(* POU STP, ST *)
PROGRAM STP
VAR
	LSL100A_MixerFloatSensor AT %I* : BOOL;
	LSH100A_MixerFloatSensor AT %I* : BOOL;
	LSH101A_EQFloatSensor AT %I* : BOOL;
	LSHH101A_EQFloatSensor AT %I* : BOOL;
	LSL101A_EQFloatSensor AT %I* : BOOL;
	LSH105A1_StreamLineFlow AT %I* : BOOL;
	LSHH105A2_StreamLineOverflow AT %I* : BOOL;
	LSL103A_SBRFloatSensor AT %I* : BOOL;
	LSHH103A_SBRFloatSensor AT %I* : BOOL;
	LSH103A_SBRFloatSensor AT %I* : BOOL;
	F100_FanStatus AT %I* : BOOL;
	D100_DoorPanelStatus AT %I* : BOOL;
	LSD101A_EQFloatSensorDry AT %I* : BOOL;
	LSD103A_SBRFloatSensorDry AT %I* : BOOL;
	XV101A1_SolenoidValveSpray_OpenStat AT %I* : BOOL;
	XV101A2_SolenoidValveSpray_OpenStat AT %I* : BOOL;
	XV102A1_ContinuosValveWater_OpenStat AT %I* : BOOL;
	XV100A1_GritRemovalValve_OpenStat AT %I* : BOOL;
	XV100A2_GritRemovalValve_OpenStat AT %I* : BOOL;
	PS101A1_Penstock_OpenStat AT %I* : BOOL;
	PS101A2_Penstock_OpenStat AT %I* : BOOL;
	PS101A1_Penstock_CloseStat AT %I* : BOOL;
	PS101A2_Penstock_CloseStat AT %I* : BOOL;
	XV101A1_SolenoidValveSpray_CloseStat AT %I* : BOOL;
	XV101A2_SolenoidValveSpray_CloseStat AT %I* : BOOL;
	XV102A1_ContinuosValveWater_CloseStat AT %I* : BOOL;
	XV100A1_GritRemovalValve_CloseStat AT %I* : BOOL;
	XV100A2_GritRemovalValve_CloseStat AT %I* : BOOL;
	M101A1_EQMixer_OverloadStat AT %I* : BOOL;
	M101A1_EQMixer_IncompleteStat AT %I* : BOOL;
	M101A2_EQMixer_OverloadStat AT %I* : BOOL;
	M101A2_EQMixer_IncompleteStat AT %I* : BOOL;
	P101A1_EQPump_OverloadStat AT %I* : BOOL;
	P101A1_EQPump_IncompleteStat AT %I* : BOOL;
	P101A2_EQPump_OverloadStat AT %I* : BOOL;
	P101A2_EQPump_IncompleteStat AT %I* : BOOL;
	PS101A1_Penstock_TripStat AT %I* : BOOL;
	PS101A2_Penstock_TripStat AT %I* : BOOL;
	F101A1_FineScr_OverloadStat AT %I* : BOOL;
	F101A2_FineScr_OverloadStat AT %I* : BOOL;
	C102A_ScreeningConveyer_OverloadStat AT %I* : BOOL;
	C101A_ScreeningCompactor_OverloadStat AT %I* : BOOL;
	C103A_GritClassifier_OverloadStat AT %I* : BOOL;
	P102A1_SBRTransferPump_OverloadStat AT %I* : BOOL;
	P102A1_SBRTransferPump_IncompleteStat AT %I* : BOOL;
	P102A2_SBRTransferPump_OverloadStat AT %I* : BOOL;
	P102A2_SBRTransferPump_IncompleteStat AT %I* : BOOL;
	M101A1_EQMixer_LocalRemoteStat AT %I* : BOOL;
	M101A2_EQMixer_LocalRemoteStat AT %I* : BOOL;
	P101A1_EQPump_LocalRemoteStat AT %I* : BOOL;
	P101A2_EQPump_LocalRemoteStat AT %I* : BOOL;
	F101A1_FineScr_LocalRemoteStat AT %I* : BOOL;
	F101A2_FineScr_LocalRemoteStat AT %I* : BOOL;
	C102A_ScreenConveyer_LocalRemoteStat AT %I* : BOOL;
	C101A_ScreenCompactor_LocalRemoteStat AT %I* : BOOL;
	C103A_GritClasifier_LocalRemoteStat AT %I* : BOOL;
	P102A1_SBRTransferPump_LocalRemoteStat AT %I* : BOOL;
	P102A2_SBRTransferPump_LocalRemoteStat AT %I* : BOOL;
	PS101A1_Penstock_LocalRemoteStat AT %I* : BOOL;
	PS101A2_Penstock_LocalRemoteStat AT %I* : BOOL;
	M101A1_EQMixer_RunStat AT %I* : BOOL;
	M101A2_EQMixer_RunStat AT %I* : BOOL;
	P101A1_EQPump_RunStat AT %I* : BOOL;
	P101A2_EQPump_RunStat AT %I* : BOOL;
	F101A1_FineScr_RunStat AT %I* : BOOL;
	F101A2_FineScr_RunStat AT %I* : BOOL;
	C102A_ScreenConveyer_RunStat AT %I* : BOOL;
	C101A_ScreenCompactor_RunStat AT %I* : BOOL;
	C103A_GritClasifier_RunStat AT %I* : BOOL;
	P102A1_SBRTransferPump_RunStat AT %I* : BOOL;
	P102A2_SBRTransferPump_RunStat AT %I* : BOOL;
	M101A1_EQMixer_EStopStat AT %I* : BOOL;
	M101A2_EQMixer_EStopStat AT %I* : BOOL;
	P101A1_EQPump_EStopStat AT %I* : BOOL;
	P101A2_EQPump_EStopStat AT %I* : BOOL;
	F101A1_FineScr_EStopStat AT %I* : BOOL;
	F101A2_FineScr_EStopStat AT %I* : BOOL;
	C102A_ScreenConveyer_EStopStat AT %I* : BOOL;
	C101A_ScreenCompactor_EStopStat AT %I* : BOOL;
	C103A_GritClasifier_EStopStat AT %I* : BOOL;
	P102A1_SBRTransferPump_EStopStat AT %I* : BOOL;
	P102A2_SBRTransferPump_EStopStat AT %I* : BOOL;
	B101A1_AirBlower_OverloadStat AT %I* : BOOL;
	B101A1_AirBlower_IncompleteStat AT %I* : BOOL;
	B101A2_AirBlower_OverloadStat AT %I* : BOOL;
	B101A2_AirBlower_IncompleteStat AT %I* : BOOL;
	B101A1_AirBlower_LocalRemoteStat AT %I* : BOOL;
	B101A2_AirBlower_LocalRemoteStat AT %I* : BOOL;
	B101A1_AirBlower_OnOffStat AT %I* : BOOL;
	B101A2_AirBlower_OnOffStat AT %I* : BOOL;
	B101A1_AirBlower_EStopStat AT %I* : BOOL;
	B101A2_AirBlower_EStopStat AT %I* : BOOL;
	XV101A1_SolenoidValveSpray_OpenCmd AT %Q* : BOOL;
	XV101A2_SolenoidValveSpray_OpenCmd AT %Q* : BOOL;
	XV102A1_ContinuosValveWater_OpenCmd AT %Q* : BOOL;
	F101A1_FineScr_RunCmd AT %Q* : BOOL;
	F101A2_FineScr_RunCmd AT %Q* : BOOL;
	C102A_ScreenConveyer_RunCmd AT %Q* : BOOL;
	C101A_ScreenCompactor_RunCmd AT %Q* : BOOL;
	C103A_GritClasifier_RunCmd AT %Q* : BOOL;
	PS101A1_Penstock_OpenCmd AT %Q* : BOOL;
	PS101A1_Penstock_CloseCmd AT %Q* : BOOL;
	PS101A2_Penstock_OpenCmd AT %Q* : BOOL;
	PS101A2_Penstock_CloseCmd AT %Q* : BOOL;
	XV100A1_GritRemovalValve_OpenCmd AT %Q* : BOOL;
	XV100A2_GritRemovalValve_OpenCmd AT %Q* : BOOL;
	P101A1_EQPump_RunCmd AT %Q* : BOOL;
	P101A2_EQPump_RunCmd AT %Q* : BOOL;
	M101A1_EQMixer_RunCmd AT %Q* : BOOL;
	M101A2_EQMixer_RunCmd AT %Q* : BOOL;
	B101A1_AirBlower_RunCmd AT %Q* : BOOL;
	B101A2_AirBlower_RunCmd AT %Q* : BOOL;
	P102A1_SBRTransferPump_RunCmd AT %Q* : BOOL;
	P102A2_SBRTransferPump_RunCmd AT %Q* : BOOL;
	AUX101A_EQFloatSensor_AlarmS1 AT %Q* : BOOL;
	AUX104A_SBRFloatSensor_AlarmS1 AT %Q* : BOOL;
	AUX105A_StreamSensorOverflow_AlarmS1 AT %Q* : BOOL;
	AUX106_CommonAlarm AT %Q* : BOOL;
	AUX107_PLCRunStat AT %Q* : BOOL;
	LSL100B_MixerFloatSensor AT %I* : BOOL;
	LSH100B_MixerFloatSensor AT %I* : BOOL;
	LSH101B_EQFloatSensor AT %I* : BOOL;
	LSHH101B_EQFloatSensor AT %I* : BOOL;
	LSL101B_EQFloatSensor AT %I* : BOOL;
	LSH105B1_StreamLineFlow AT %I* : BOOL;
	LSHH105B2_StreamLineOverflow AT %I* : BOOL;
	LSH103B_SBRFloatSensor AT %I* : BOOL;
	LSHH103B_SBRFloatSensor AT %I* : BOOL;
	LSL103B_SBRFloatSensor AT %I* : BOOL;
	LSD101B_EQFloatSensorDry AT %I* : BOOL;
	LSD103B_SBRFloatSensorDry AT %I* : BOOL;
	XV101B1_SolenoidValveSpray_OpenStat AT %I* : BOOL;
	XV101B2_SolenoidValveSpray_OpenStat AT %I* : BOOL;
	XV102B1_ContinuosValveWater_OpenStat AT %I* : BOOL;
	XV100B1_GritRemovalValve_OpenStat AT %I* : BOOL;
	XV100B2_GritRemovalValve_OpenStat AT %I* : BOOL;
	PS101B1_Penstock_OpenStat AT %I* : BOOL;
	PS101B2_Penstock_OpenStat AT %I* : BOOL;
	PS101B1_Penstock_CloseStat AT %I* : BOOL;
	PS101B2_Penstock_CloseStat AT %I* : BOOL;
	XV101B1_SolenoidValveSpray_CloseStat AT %I* : BOOL;
	XV101B2_SolenoidValveSpray_CloseStat AT %I* : BOOL;
	XV102B1_ContinuosValveWater_CloseStat AT %I* : BOOL;
	XV100B1_GritRemovalValve_CloseStat AT %I* : BOOL;
	XV100B2_GritRemovalValve_CloseStat AT %I* : BOOL;
	M101B1_EQMixer_OverloadStat AT %I* : BOOL;
	M101B1_EQMixer_IncompleteStat AT %I* : BOOL;
	M101B2_EQMixer_OverloadStat AT %I* : BOOL;
	M101B2_EQMixer_IncompleteStat AT %I* : BOOL;
	P101B1_EQPump_OverloadStat AT %I* : BOOL;
	P101B1_EQPump_IncompleteStat AT %I* : BOOL;
	P101B2_EQPump_OverloadStat AT %I* : BOOL;
	P101B2_EQPump_IncompleteStat AT %I* : BOOL;
	PS101B1_Penstock_TripStat AT %I* : BOOL;
	PSB101B2_Penstock_TripStat AT %I* : BOOL;
	F101B1_FineScr_OverloadStat AT %I* : BOOL;
	F101B2_FineScr_OverloadStat AT %I* : BOOL;
	C102B_ScreeningConveyer_OverloadStat AT %I* : BOOL;
	C101B_ScreeningCompactor_OverloadStat AT %I* : BOOL;
	C103B_GritClassifier_OverloadStat AT %I* : BOOL;
	P102B1_SBRTransferPump_OverloadStat AT %I* : BOOL;
	P102B1_SBRTransferPump_IncompleteStat AT %I* : BOOL;
	P102B2_SBRTransferPump_OverloadStat AT %I* : BOOL;
	P102B2_SBRTransferPump_IncompleteStat AT %I* : BOOL;
	M101B1_EQMixer_LocalRemoteStat AT %I* : BOOL;
	M101B2_EQMixer_LocalRemoteStat AT %I* : BOOL;
	P101B1_EQPump_LocalRemoteStat AT %I* : BOOL;
	P101B2_EQPump_LocalRemoteStat AT %I* : BOOL;
	F101B1_FineScr_LocalRemoteStat AT %I* : BOOL;
	F101B2_FineScr_LocalRemoteStat AT %I* : BOOL;
	C102B_ScreenConveyer_LocalRemoteStat AT %I* : BOOL;
	C101B_ScreenCompactor_LocalRemoteStat AT %I* : BOOL;
	C103B_GritClasifiier_LocalRemoteStat AT %I* : BOOL;
	P102B1_SBRTransferPump_LocalRemoteStat AT %I* : BOOL;
	P102B2_SBRTransferPump_LocalRemoteStat AT %I* : BOOL;
	PS101B1_Penstock_LocalRemoteStat AT %I* : BOOL;
	PS101B2_Penstock_LocalRemoteStat AT %I* : BOOL;
	M101B1_EQMixer_RunStat AT %I* : BOOL;
	M101B2_EQMixer_RunStat AT %I* : BOOL;
	P101B1_EQPump_RunStat AT %I* : BOOL;
	P101B2_EQPump_RunStat AT %I* : BOOL;
	F101B1_FineScr_RunStat AT %I* : BOOL;
	F101B2_FineScr_RunStat AT %I* : BOOL;
	C102B_ScreenConveyer_RunStat AT %I* : BOOL;
	C101B_ScreenCompactor_RunStat AT %I* : BOOL;
	C103B_GritClasifier_RunStat AT %I* : BOOL;
	P102B1_SBRTransferPump_RunStat AT %I* : BOOL;
	P102B2_SBRTransferPump_RunStat AT %I* : BOOL;
	M101B1_EQMixer_EStopStat AT %I* : BOOL;
	M101B2_EQMixer_EStopStat AT %I* : BOOL;
	P101B1_EQPump_EStopStat AT %I* : BOOL;
	P101B2_EQPump_EStopStat AT %I* : BOOL;
	F101B1_FineScr_EStopStat AT %I* : BOOL;
	F101B2_FineScr_EStopStat AT %I* : BOOL;
	C102B_ScreenConveyer_EStopStat AT %I* : BOOL;
	C101B_ScreenCompactor_EStopStat AT %I* : BOOL;
	C103B_GritClasifier_EStopStat AT %I* : BOOL;
	P102B1_SBRTransferPump_EStopStat AT %I* : BOOL;
	P102B2_SBRTransferPump_EStopStat AT %I* : BOOL;
	VE801A_SuctionFan_OnOffStat AT %I* : BOOL;
	P802A_CirculationPump_OnOffStat AT %I* : BOOL;
	P803A_CirculationPump_OnOffStat AT %I* : BOOL;
	P804A_CirculationPump_OnOffStat AT %I* : BOOL;
	P805A1_H2S04Pump_OnOffStat AT %I* : BOOL;
	P805A2_H2S04Pump_OnOffStat AT %I* : BOOL;
	P806A1_NAOHPump_OnOffStat AT %I* : BOOL;
	P806A2_NAOHPump_OnOffStat AT %I* : BOOL;
	P807A1_NAOCLPump_OnOffStat AT %I* : BOOL;
	P807A2_NAOCLPump_OnOffStat AT %I* : BOOL;
	VE801A_SuctionFan_OverloadStat AT %I* : BOOL;
	P802A_CirculationPump_OverloadStat AT %I* : BOOL;
	P803A_CirculationPump_OverloadStat AT %I* : BOOL;
	P804A_CirculationPump_OverloadStat AT %I* : BOOL;
	P805A1_H2S04Pump_OverloadStat AT %I* : BOOL;
	P805A2_H2S04Pump_OverloadStat AT %I* : BOOL;
	P806A1_NAOHPump_OverloadStat AT %I* : BOOL;
	P806A2_NAOHPump_OverloadStat AT %I* : BOOL;
	P807A1_NAOCLPump_OverloadStat AT %I* : BOOL;
	P807A2_NAOCLPump_OverloadStat AT %I* : BOOL;
	VE801A_SuctionFan_EStopStat AT %I* : BOOL;
	P802A_CirculationPump_EStopStat AT %I* : BOOL;
	P803A_CirculationPump_EStopStat AT %I* : BOOL;
	P804A_CirculationPump_EStopStat AT %I* : BOOL;
	P805A1_H2S04Pump_EStopStat AT %I* : BOOL;
	P805A2_H2S04Pump_EStopStat AT %I* : BOOL;
	P806A1_NAOHPump_EStopStat AT %I* : BOOL;
	P806A2_NAOHPump_EStopStat AT %I* : BOOL;
	P807A1_NAOCLPump_EStopStat AT %I* : BOOL;
	P807A2_NAOCLPump_EStopStat AT %I* : BOOL;
	XV101B1_SolenoidValveSpray_OpenCmd AT %Q* : BOOL;
	XV101B2_SolenoidValveSpray_OpenCmd AT %Q* : BOOL;
	XV102B1_ContinuosValveWater_OpenCmd AT %Q* : BOOL;
	F101B1_FineScr_RunCmd AT %Q* : BOOL;
	F101B2_FineScr_RunCmd AT %Q* : BOOL;
	C102B_ScreenConveyer_RunCmd AT %Q* : BOOL;
	C101B_ScreenCompactor_RunCmd AT %Q* : BOOL;
	C103B_GritClasifier_RunCmd AT %Q* : BOOL;
	PS101B1_Penstock_OpenCmd AT %Q* : BOOL;
	PS101B1_Penstock_CloseCmd AT %Q* : BOOL;
	PS101B2_Penstock_OpenCmd AT %Q* : BOOL;
	PS101B2_Penstock_CloseCmd AT %Q* : BOOL;
	XV100B1_GritRemovalValve_OpenCmd AT %Q* : BOOL;
	XV100B2_GritRemovalValve_OpenCmd AT %Q* : BOOL;
	P101B1_EQPump_RunCmd AT %Q* : BOOL;
	P101B2_EQPump_RunCmd AT %Q* : BOOL;
	M101B1_EQMixer_RunCmd AT %Q* : BOOL;
	M101B2_EQMixer_RunCmd AT %Q* : BOOL;
	P102B1_SBRTransferPump_RunCmd AT %Q* : BOOL;
	P102B2_SBRTransferPump_RunCmd AT %Q* : BOOL;
	AUX101B_EQFloatSensor_AlarmS2 AT %Q* : BOOL;
	AUX104B_SBRFloatSensor_AlarmS2 AT %Q* : BOOL;
	AUX105B_StreamSensorOverflow_AlarmS2 AT %Q* : BOOL;
	F200A_FanStatus AT %I* : BOOL;
	D200A_DoorPanelStatus AT %I* : BOOL;
	XV261A_DecanterR1_OverloadStat AT %I* : BOOL;
	XV262A_DecanterR2_OverloadStat AT %I* : BOOL;
	XV263A_DecanterR3_OverloadStat AT %I* : BOOL;
	XV264A_DecanterR4_OverloadStat AT %I* : BOOL;
	M200A1A_MixerR1_RunStat AT %I* : BOOL;
	M200A1B_MixerR1_RunStat AT %I* : BOOL;
	M200A1C_MixerR1_RunStat AT %I* : BOOL;
	M200A2A_MixerR2_RunStat AT %I* : BOOL;
	M200A2B_MixerR2_RunStat AT %I* : BOOL;
	M200A2C_MixerR2_RunStat AT %I* : BOOL;
	M200A3A_MixerR3_RunStat AT %I* : BOOL;
	M200A3B_MixerR3_RunStat AT %I* : BOOL;
	M200A3C_MixerR3_RunStat AT %I* : BOOL;
	M200A4A_MixerR4_RunStat AT %I* : BOOL;
	M200A4B_MixerR4_RunStat AT %I* : BOOL;
	M200A4C_MixerR4_RunStat AT %I* : BOOL;
	B201A1_AirBlowerS1_RunStat AT %I* : BOOL;
	B201A2_AirBlowerS1_RunStat AT %I* : BOOL;
	B201A3_AirBlowerS1_RunStat AT %I* : BOOL;
	M200A1A_MixerR1_LocalRemoteStat AT %I* : BOOL;
	M200A1B_MixerR1_LocalRemoteStat AT %I* : BOOL;
	M200A1C_MixerR1_LocalRemoteStat AT %I* : BOOL;
	M200A2A_MixerR2_LocalRemoteStat AT %I* : BOOL;
	M200A2B_MixerR2_LocalRemoteStat AT %I* : BOOL;
	M200A2C_MixerR2_LocalRemoteStat AT %I* : BOOL;
	M200A3A_MixerR3_LocalRemoteStat AT %I* : BOOL;
	M200A3B_MixerR3_LocalRemoteStat AT %I* : BOOL;
	M200A3C_MixerR3_LocalRemoteStat AT %I* : BOOL;
	M200A4A_MixerR4_LocalRemoteStat AT %I* : BOOL;
	M200A4B_MixerR4_LocalRemoteStat AT %I* : BOOL;
	M200A4C_MixerR4_LocalRemoteStat AT %I* : BOOL;
	B201A1_AirBlowerS1_LocalRemoteStat AT %I* : BOOL;
	B201A2_AirBlowerS1_LocalRemoteStat AT %I* : BOOL;
	B201A3_AirBlowerS1_LocalRemoteStat AT %I* : BOOL;
	XV261A_DecanterR1_LocalRemoteStat AT %I* : BOOL;
	XV262A_DecanterR2_LocalRemoteStat AT %I* : BOOL;
	XV263A_DecanterR3_LocalRemoteStat AT %I* : BOOL;
	XV264A_DecanterR4_LocalRemoteStat AT %I* : BOOL;
	P201A1_DesludgePumpS1_LocalRemoteStat AT %I* : BOOL;
	P201A2_DesludgePumpS1_LocalRemoteStat AT %I* : BOOL;
	P201A1_DesludgePumpS1_RunStat AT %I* : BOOL;
	P201A2_DesludgePumpS1_RunStat AT %I* : BOOL;
	M200A1A_MixerR1_OverloadStat AT %I* : BOOL;
	M200A1A_MixerR1_IncompleteStat AT %I* : BOOL;
	M200A1B_MixerR1_OverloadStat AT %I* : BOOL;
	M200A1B_MixerR1_IncompleteStat AT %I* : BOOL;
	M200A1C_MixerR1_OverloadStat AT %I* : BOOL;
	M200A1C_MixerR1_IncompleteStat AT %I* : BOOL;
	M200A2A_MixerR2_OverloadStat AT %I* : BOOL;
	M200A2A_MixerR2_IncompleteStat AT %I* : BOOL;
	M200A2B_MixerR2_OverloadStat AT %I* : BOOL;
	M200A2B_MixerR2_IncompleteStat AT %I* : BOOL;
	M200A2C_MixerR2_OverloadStat AT %I* : BOOL;
	M200A2C_MixerR2_IncompleteStat AT %I* : BOOL;
	M200A3A_MixerR3_OverloadStat AT %I* : BOOL;
	M200A3A_MixerR3_IncompleteStat AT %I* : BOOL;
	M200A3B_MixerR3_OverloadStat AT %I* : BOOL;
	M200A3B_MixerR3_IncompleteStat AT %I* : BOOL;
	M200A3C_MixerR3_OverloadStat AT %I* : BOOL;
	M200A3C_MixerR3_IncompleteStat AT %I* : BOOL;
	M200A4A_MixerR4_OverloadStat AT %I* : BOOL;
	M200A4A_MixerR4_IncompleteStat AT %I* : BOOL;
	M200A4B_MixerR4_OverloadStat AT %I* : BOOL;
	M200A4B_MixerR4_IncompleteStat AT %I* : BOOL;
	M200A4C_MixerR4_OverloadStat AT %I* : BOOL;
	M200A4C_MixerR4_IncompleteStat AT %I* : BOOL;
	B201A1_AirBlowerS1_OverloadStat AT %I* : BOOL;
	B201A1_AirBlowerS1_IncompleteStat AT %I* : BOOL;
	B201A2_AirBlowerS1_OverloadStat AT %I* : BOOL;
	B201A2_AirBlowerS1_IncompleteStat AT %I* : BOOL;
	B201A3_AirBlowerS1_OverloadStat AT %I* : BOOL;
	B201A3_AirBlowerS1_IncompleteStat AT %I* : BOOL;
	P201A1_DesludgePumpS1_OverloadStatus AT %I* : BOOL;
	P201A2_DesludgePumpS1_OverloadStatus AT %I* : BOOL;
	M200A1A_MixerR1_EStopStat AT %I* : BOOL;
	M200A1B_MixerR1_EStopStat AT %I* : BOOL;
	M200A1C_MixerR1_EStopStat AT %I* : BOOL;
	M200A2A_MixerR2_EStopStat AT %I* : BOOL;
	M200A2B_MixerR2_EStopStat AT %I* : BOOL;
	M200A2C_MixerR2_EStopStat AT %I* : BOOL;
	M200A3A_MixerR3_EStopStat AT %I* : BOOL;
	M200A3B_MixerR3_EStopStat AT %I* : BOOL;
	M200A3C_MixerR3_EStopStat AT %I* : BOOL;
	M200A4A_MixerR3_EStopStat AT %I* : BOOL;
	M200A4B_MixerR3_EStopStat AT %I* : BOOL;
	M200A4C_MixerR3_EStopStat AT %I* : BOOL;
	B201A1_AirBlowerS1_EStopStat AT %I* : BOOL;
	B201A2_AirBlowerS1_EStopStat AT %I* : BOOL;
	B201A3_AirBlowerS1_EStopStat AT %I* : BOOL;
	XV261A_DecanterR1_EStopStat AT %I* : BOOL;
	XV262A_DecanterR2_EStopStat AT %I* : BOOL;
	XV263A_DecanterR3_EStopStat AT %I* : BOOL;
	XV264A_DecanterR4_EStopStat AT %I* : BOOL;
	P201A1_DesludgePumpS1_EStopStat AT %I* : BOOL;
	P201A2_DesludgePumpS1_EStopStat AT %I* : BOOL;
	XV261A_DecanterR1_FwdStat AT %I* : BOOL;
	XV262A_DecanterR2_FwdStat AT %I* : BOOL;
	XV263A_DecanterR3_FwdStat AT %I* : BOOL;
	XV264A_DecanterR4_FwdStat AT %I* : BOOL;
	XV261A_DecanterR1_RvsStat AT %I* : BOOL;
	XV262A_DecanterR2_RvsStat AT %I* : BOOL;
	XV263A_DecanterR3_RvsStat AT %I* : BOOL;
	XV264A_DecanterR4_RvsStat AT %I* : BOOL;
	FT100A_FlowTotalizerS1 : REAL;
	FT100A_FlowTotalizerS1_ScaledValue AT %I*:INT;
	M200A1A_MixerR1_RunCmd AT %Q* : BOOL;
	M200A1B_MixerR1_RunCmd AT %Q* : BOOL;
	M200A1C_MixerR1_RunCmd AT %Q* : BOOL;
	M200A2A_MixerR2_RunCmd AT %Q* : BOOL;
	M200A2B_MixerR2_RunCmd AT %Q* : BOOL;
	M200A2C_MixerR2_RunCmd AT %Q* : BOOL;
	M200A3A_MixerR3_RunCmd AT %Q* : BOOL;
	M200A3B_MixerR3_RunCmd AT %Q* : BOOL;
	M200A3C_MixerR3_RunCmd AT %Q* : BOOL;
	M200A4A_MixerR4_RunCmd AT %Q* : BOOL;
	M200A4B_MixerR4_RunCmd AT %Q* : BOOL;
	M200A4C_MixerR4_RunCmd AT %Q* : BOOL;
	XV261A_DecanterR1_FwdCmd AT %Q* : BOOL;
	XV262A_DecanterR2_FwdCmd AT %Q* : BOOL;
	XV263A_DecanterR3_FwdCmd AT %Q* : BOOL;
	XV264A_DecanterR4_FwdCmd AT %Q* : BOOL;
	XV261A_DecanterR1_RvsCmd AT %Q* : BOOL;
	XV262A_DecanterR2_RvsCmd AT %Q* : BOOL;
	XV263A_DecanterR3_RvsCmd AT %Q* : BOOL;
	XV264A_DecanterR4_RvsCmd AT %Q* : BOOL;
	B201A1_AirBlowerS1_RunCmd AT %Q* : BOOL;
	B201A2_AirBlowerS1_RunCmd AT %Q* : BOOL;
	B201A3_AirBlowerS1_RunCmd AT %Q* : BOOL;
	P201A1_DesludgePump_RunCmd AT %Q* : BOOL;
	P201A2_DesludgePump_RunCmd AT %Q* : BOOL;
	AUXA1_ReactorS1R1_OpsStat AT %Q* : BOOL;
	AUXA2_ReactorS1R2_OpsStat AT %Q* : BOOL;
	AUXA3_ReactorS1R3_OpsStat AT %Q* : BOOL;
	AUXA4_ReactorS1R4_OpsStat AT %Q* : BOOL;
	AUXB1_ReactorS2R1_OpsStat AT %Q* : BOOL;
	AUXB2_ReactorS2R2_OpsStat AT %Q* : BOOL;
	AUXB3_ReactorS2R3_OpsStat AT %Q* : BOOL;
	AUXB4_ReactorS2R4_OpsStat AT %Q* : BOOL;
	AUXA5_BlowerS1R1 AT %Q* : BOOL;
	AUXA6_BlowerS1R2 AT %Q* : BOOL;
	AUXA7_BlowerS1R3 AT %Q* : BOOL;
	AUXB5_BlowerS2R1 AT %Q* : BOOL;
	AUXB6_BlowerS2R2 AT %Q* : BOOL;
	AUXB7_BlowerS2R3 AT %Q* : BOOL;
	AUX201_CommonAlarm AT %Q* : BOOL;
	AUX202_PLCRunStat AT %Q* : BOOL;
	F200B_FanStatus AT %I* : BOOL;
	D200B_DoorPanelStatus AT %I* : BOOL;
	XV261B_DecanterR1_OverloadStat AT %I* : BOOL;
	XV262B_DecanterR2_OverloadStat AT %I* : BOOL;
	XV263B_DecanterR3_OverloadStat AT %I* : BOOL;
	XV264B_DecanterR4_OverloadStat AT %I* : BOOL;
	M200B1A_MixerR1_RunStat AT %I* : BOOL;
	M200B1B_MixerR1_RunStat AT %I* : BOOL;
	M200B1C_MixerR1_RunStat AT %I* : BOOL;
	M200B2A_MixerR2_RunStat AT %I* : BOOL;
	M200B2B_MixerR2_RunStat AT %I* : BOOL;
	M200B2C_MixerR2_RunStat AT %I* : BOOL;
	M200B3A_MixerR3_RunStat AT %I* : BOOL;
	M200B3B_MixerR3_RunStat AT %I* : BOOL;
	M200B3C_MixerR3_RunStat AT %I* : BOOL;
	M200B4A_MixerR4_RunStat AT %I* : BOOL;
	M200B4B_MixerR4_RunStat AT %I* : BOOL;
	M200B4C_MixerR4_RunStat AT %I* : BOOL;
	B201B1_AirBlowerS2_RunStat AT %I* : BOOL;
	B201B2_AirBlowerS2_RunStat AT %I* : BOOL;
	B201B3_AirBlowerS2_RunStat AT %I* : BOOL;
	M200B1A_MixerR1_LocalRemoteStat AT %I* : BOOL;
	M200B1B_MixerR1_LocalRemoteStat AT %I* : BOOL;
	M200B1C_MixerR1_LocalRemoteStat AT %I* : BOOL;
	M200B2A_MixerR2_LocalRemoteStat AT %I* : BOOL;
	M200B2B_MixerR2_LocalRemoteStat AT %I* : BOOL;
	M200B2C_MixerR2_LocalRemoteStat AT %I* : BOOL;
	M200B3A_MixerR3_LocalRemoteStat AT %I* : BOOL;
	M200B3B_MixerR3_LocalRemoteStat AT %I* : BOOL;
	M200B3C_MixerR3_LocalRemoteStat AT %I* : BOOL;
	M200B4A_MixerR4_LocalRemoteStat AT %I* : BOOL;
	M200B4B_MixerR4_LocalRemoteStat AT %I* : BOOL;
	M200B4C_MixerR4_LocalRemoteStat AT %I* : BOOL;
	B201B1_AirBlowerS2_LocalRemoteStat AT %I* : BOOL;
	B201B2_AirBlowerS2_LocalRemoteStat AT %I* : BOOL;
	B201B3_AirBlowerS2_LocalRemoteStat AT %I* : BOOL;
	XV261B_DecanterR1_LocalRemoteStat AT %I* : BOOL;
	XV262B_DecanterR2_LocalRemoteStat AT %I* : BOOL;
	XV263B_DecanterR3_LocalRemoteStat AT %I* : BOOL;
	XV264B_DecanterR4_LocalRemoteStat AT %I* : BOOL;
	P201B1_DesludgePumpS2_LocalRemoteStat AT %I* : BOOL;
	P201B2_DesludgePumpS2_LocalRemoteStat AT %I* : BOOL;
	P201B1_DesludgePumpS2_RunStat AT %I* : BOOL;
	P201B2_DesludgePumpS2_RunStat AT %I* : BOOL;
	M200B1A_MixerR1_OverloadStat AT %I* : BOOL;
	M200B1A_MixerR1_IncompleteStat AT %I* : BOOL;
	M200B1B_MixerR1_OverloadStat AT %I* : BOOL;
	M200B1B_MixerR1_IncompleteStat AT %I* : BOOL;
	M200B1C_MixerR1_OverloadStat AT %I* : BOOL;
	M200B1C_MixerR1_IncompleteStat AT %I* : BOOL;
	M200B2A_MixerR2_OverloadStat AT %I* : BOOL;
	M200B2A_MixerR2_IncompleteStat AT %I* : BOOL;
	M200B2B_MixerR2_OverloadStat AT %I* : BOOL;
	M200B2B_MixerR2_IncompleteStat AT %I* : BOOL;
	M200B2C_MixerR2_OverloadStat AT %I* : BOOL;
	M200B2C_MixerR2_IncompleteStat AT %I* : BOOL;
	M200B3A_MixerR3_OverloadStat AT %I* : BOOL;
	M200B3A_MixerR2_IncompleteStat AT %I* : BOOL;
	M200B3B_MixerR3_OverloadStat AT %I* : BOOL;
	M200B3B_MixerR3_IncompleteStat AT %I* : BOOL;
	M200B3C_MixerR3_OverloadStat AT %I* : BOOL;
	M200B3C_MixerR3_IncompleteStat AT %I* : BOOL;
	M200B4A_MixerR4_OverloadStat AT %I* : BOOL;
	M200B4A_MixerR4_IncompleteStat AT %I* : BOOL;
	M200B4B_MixerR4_OverloadStat AT %I* : BOOL;
	M200B4B_MixerR4_IncompleteStat AT %I* : BOOL;
	M200B4C_MixerR4_OverloadStat AT %I* : BOOL;
	M200B4C_MixerR4_IncompleteStat AT %I* : BOOL;
	B201B1_AirBlowerS2_OverloadStat AT %I* : BOOL;
	B201B1_AirBlowerS2_IncompleteStat AT %I* : BOOL;
	B201B2_AirBlowerS2_OverloadStat AT %I* : BOOL;
	B201B2_AirBlowerS2_IncompleteStat AT %I* : BOOL;
	B201B3_AirBlowerS2_OverloadStat AT %I* : BOOL;
	B201B3_AirBlowerS2_IncompleteStat AT %I* : BOOL;
	P201B1_DesludgePumpS2_OverloadStat AT %I* : BOOL;
	P201B2_DesludgePumpS2_OverloadStat AT %I* : BOOL;
	M200B1A_MixerR1_EStopStat AT %I* : BOOL;
	M200B1B_MixerR1_EStopStat AT %I* : BOOL;
	M200B1C_MixerR1_EStopStat AT %I* : BOOL;
	M200B2A_MixerR2_EStopStat AT %I* : BOOL;
	M200B2B_MixerR2_EStopStat AT %I* : BOOL;
	M200B2C_MixerR2_EStopStat AT %I* : BOOL;
	M200B3A_MixerR3_EStopStat AT %I* : BOOL;
	M200B3B_MixerR3_EStopStat AT %I* : BOOL;
	M200B3C_MixerR3_EStopStat AT %I* : BOOL;
	M200B4A_MixerR4_EStopStat AT %I* : BOOL;
	M200B4B_MixerR4_EStopStat AT %I* : BOOL;
	M200B4C_MixerR4_EStopStat AT %I* : BOOL;
	B201B1_AirBlowerS2_EStopStat AT %I* : BOOL;
	B201B2_AirBlowerS2_EStopStat AT %I* : BOOL;
	B201B3_AirBlowerS2_EStopStat AT %I* : BOOL;
	XV261B_DecanterR1_EStopStat AT %I* : BOOL;
	XV262B_DecanterR2_EStopStat AT %I* : BOOL;
	XV263B_DecanterR3_EStopStat AT %I* : BOOL;
	XV264B_DecanterR4_EStopStat AT %I* : BOOL;
	P201B1_DesludgePumpS2_EStopStat AT %I* : BOOL;
	P201B2_DesludgePumpS2_EStopStat AT %I* : BOOL;
	XV261B_DecanterR1_FwdStat AT %I* : BOOL;
	XV262B_DecanterR2_FwdStat AT %I* : BOOL;
	XV263B_DecanterR3_FwdStat AT %I* : BOOL;
	XV264B_DecanterR4_FwdStat AT %I* : BOOL;
	XV261B_DecanterR1_RvsStat AT %I* : BOOL;
	XV262B_DecanterR2_RvsStat AT %I* : BOOL;
	XV263B_DecanterR3_RvsStat AT %I* : BOOL;
	XV264B_DecanterR4_RvsStat AT %I* : BOOL;
	FT100B_FlowTotalizerS2 : REAL;
	FT100B_FlowTotalizerS2_ScaledValue AT %I*:INT;
	M200B1A_MixerR1_RunCmd AT %Q* : BOOL;
	M200B1B_MixerR1_RunCmd AT %Q* : BOOL;
	M200B1C_MixerR1_RunCmd AT %Q* : BOOL;
	M200B2A_MixerR2_RunCmd AT %Q* : BOOL;
	M200B2B_MixerR2_RunCmd AT %Q* : BOOL;
	M200B2C_MixerR2_RunCmd AT %Q* : BOOL;
	M200B3A_MixerR3_RunCmd AT %Q* : BOOL;
	M200B3B_MixerR3_RunCmd AT %Q* : BOOL;
	M200B3C_MixerR3_RunCmd AT %Q* : BOOL;
	M200B4A_MixerR4_RunCmd AT %Q* : BOOL;
	M200B4B_MixerR4_RunCmd AT %Q* : BOOL;
	M200B4C_MixerR4_RunCmd AT %Q* : BOOL;
	XV261B_DecanterR1_FwdCmd AT %Q* : BOOL;
	XV262B_DecanterR2_FwdCmd AT %Q* : BOOL;
	XV263B_DecanterR3_FwdCmd AT %Q* : BOOL;
	XV264B_DecanterR4_FwdCmd AT %Q* : BOOL;
	XV261B_DecanterR1_RvsCmd AT %Q* : BOOL;
	XV262B_DecanterR2_RvsCmd AT %Q* : BOOL;
	XV263B_DecanterR3_RvsCmd AT %Q* : BOOL;
	XV264B_DecanterR4_RvsCmd AT %Q* : BOOL;
	B201B1_AirBlowerS2_RunCmd AT %Q* : BOOL;
	B201B2_AirBlowerS2_RunCmd AT %Q* : BOOL;
	B201B3_AirBlowerS2_RunCmd AT %Q* : BOOL;
	P201B1_DesludgePumpS2_RunCmd AT %Q* : BOOL;
	P201B2_DesludgePumpS2_RunCmd AT %Q* : BOOL;
	LSH201A1_LevelSensorR1 AT %I* : BOOL;
	LSH201A2_LevelSensorR2 AT %I* : BOOL;
	LSH201A3_LevelSensorR3 AT %I* : BOOL;
	LSH201A4_LevelSensorR4 AT %I* : BOOL;
	OPR1A_ReactorStatus AT %I* : BOOL;
	OPR2A_ReactorStatus AT %I* : BOOL;
	OPR3A_ReactorStatus AT %I* : BOOL;
	OPR4A_ReactorStatus AT %I* : BOOL;
	D201A_DoorPanelStatus AT %I* : BOOL;
	F201A_FanStatus AT %I* : BOOL;
	HR201A1_DecantHighLevelR1 AT %I* : BOOL;
	LR201A1_DecantLowLevelR1 AT %I* : BOOL;
	HR201A2_DecantHighLevelR2 AT %I* : BOOL;
	LR201A2_DecantLowLevelR2 AT %I* : BOOL;
	HR201A3_DecantHighLevelR3 AT %I* : BOOL;
	LR201A3_DecantLowLevelR3 AT %I* : BOOL;
	HR201A4_DecantHighLevelR4 AT %I* : BOOL;
	LR201A4_DecantLowLevelR4 AT %I* : BOOL;
	XV205A_SBRValveR1_OpenStat AT %I* : BOOL;
	XV206A_SBRValveR2_OpenStat AT %I* : BOOL;
	XV207A_SBRValveR3_OpenStat AT %I* : BOOL;
	XV208A_SBRValveR4_OpenStat AT %I* : BOOL;
	XV201A_AirBlowerValveR1_OpenStat AT %I* : BOOL;
	XV202A_AirBlowerValveR2_OpenStat AT %I* : BOOL;
	XV203A_AirBlowerValveR3_OpenStat AT %I* : BOOL;
	XV204A_AirBlowerValveR4_OpenStat AT %I* : BOOL;
	XV221A_LimeValveR1_OpenStat AT %I* : BOOL;
	XV222A_LimeValveR2_OpenStat AT %I* : BOOL;
	XV223A_LimeValveR3_OpenStat AT %I* : BOOL;
	XV224A_LimeValveR4_OpenStat AT %I* : BOOL;
	XV211A_AlumValveR1_OpenStat AT %I* : BOOL;
	XV212A_AlumValveR2_OpenStat AT %I* : BOOL;
	XV213A_AlumValveR3_OpenStat AT %I* : BOOL;
	XV214A_AlumValveR4_OpenStat AT %I* : BOOL;
	XV205A_SBRValveR1_CloseStat AT %I* : BOOL;
	XV206A_SBRValveR2_CloseStat AT %I* : BOOL;
	XV207A_SBRValveR3_CloseStat AT %I* : BOOL;
	XV208A_SBRValveR4_CloseStat AT %I* : BOOL;
	XV201A_AirBlowerValveR1_CloseStat AT %I* : BOOL;
	XV202A_AirBlowerValveR2_CloseStat AT %I* : BOOL;
	XV203A_AirBlowerValveR3_CloseStat AT %I* : BOOL;
	XV204A_AirBlowerValveR4_CloseStat AT %I* : BOOL;
	XV221A_LimeValveR1_CloseStat AT %I* : BOOL;
	XV222A_LimeValveR2_CloseStat AT %I* : BOOL;
	XV223A_LimeValveR3_CloseStat AT %I* : BOOL;
	XV224A_LimeValveR4_CloseStat AT %I* : BOOL;
	XV211A_AlumValveR1_CloseStat AT %I* : BOOL;
	XV212A_AlumValveR2_CloseStat AT %I* : BOOL;
	XV213A_AlumValveR3_CloseStat AT %I* : BOOL;
	XV214A_AlumValveR4_CloseStat AT %I* : BOOL;
	XV241A_SludgeValveR1_CloseStat AT %I* : BOOL;
	XV242A_SludgeValveR2_CloseStat AT %I* : BOOL;
	XV243A_SludgeValveR3_CloseStat AT %I* : BOOL;
	XV244A_SludgeValveR4_CloseStat AT %I* : BOOL;
	XV241A_SludgeValveR1_OpenStat AT %I* : BOOL;
	XV242A_SludgeValveR2_OpenStat AT %I* : BOOL;
	XV243A_SludgeValveR3_OpenStat AT %I* : BOOL;
	XV244A_SludgeValveR4_OpenStat AT %I* : BOOL;
	D0201A4_DOProfilesR4 : REAL;
	D0201A4_DOProfilesR4_ScaledValue AT %I*:INT;
	DO201A1_DOProfilesR1:REAL;
	DO201A1_DOProfilesR1_ScaledValue AT %I*:INT;
	DO201A2_DOProfilesR2 :REAL;
	DO201A2_DOProfilesR2_ScaledValue AT %I*:INT;
	DO201A3_DOProfilesR3 :REAL;
	DO201A3_DOProfilesR3_ScaledValue AT %I*:INT;
	PHT201A1_pHlevelR1 : REAL;
	PHT201A1_pHlevelR1_ScaledValue AT %I*:INT;
	PHT201A2_pHlevelR2 : REAL;
	PHT201A2_pHlevelR2_ScaledValue AT %I*:INT;
	PHT201A3_pHlevelR3 : REAL;
	PHT201A3_pHlevelR3_ScaledValue AT %I*:INT;
	PHT201A4_pHlevelR4 : REAL;
	PHT201A4_pHlevelR4_ScaledValue AT %I*:INT;
	XV205A_SBRValveR1_OpenCmd AT %Q* : BOOL;
	XV206A_SBRValveR2_OpenCmd AT %Q* : BOOL;
	XV207A_SBRValveR3_OpenCmd AT %Q* : BOOL;
	XV208A_SBRValveR4_OpenCmd AT %Q* : BOOL;
	XV201A_AirBlowerValveR1_OpenCmd AT %Q* : BOOL;
	XV202A_AirBlowerValveR2_OpenCmd AT %Q* : BOOL;
	XV203A_AirBlowerValveR3_OpenCmd AT %Q* : BOOL;
	XV204A_AirBlowerValveR4_OpenCmd AT %Q* : BOOL;
	XV221A_LimeValveR1_OpenCmd AT %Q* : BOOL;
	XV222A_LimeValveR2_OpenCmd AT %Q* : BOOL;
	XV223A_LimeValveR3_OpenCmd AT %Q* : BOOL;
	XV224A_LimeValveR4_OpenCmd AT %Q* : BOOL;
	XV211A_AlumValveR1_OpenCmd AT %Q* : BOOL;
	XV212A_AlumValveR2_OpenCmd AT %Q* : BOOL;
	XV213A_AlumValveR3_OpenCmd AT %Q* : BOOL;
	XV214A_AlumValveR4_OpenCmd AT %Q* : BOOL;
	XV241A_SludgeValveR1_OpenCmd AT %Q* : BOOL;
	XV242A_SludgeValveR2_OpenCmd AT %Q* : BOOL;
	XV243A_SludgeValveR3_OpenCmd AT %Q* : BOOL;
	XV244A_SludgeValveR4_OpenCmd AT %Q* : BOOL;
	XV241A_SludgeValveR1_CloseCmd AT %Q* : BOOL;
	XV242A_SludgeValveR2_CloseCmd AT %Q* : BOOL;
	XV243A_SludgeValveR3_CloseCmd AT %Q* : BOOL;
	XV244A_SludgeValveR4_CloseCmd AT %Q* : BOOL;
	XV205A_SBRValveR1_CloseCmd AT %Q* : BOOL;
	XV206A_SBRValveR2_CloseCmd AT %Q* : BOOL;
	XV207A_SBRValveR3_CloseCmd AT %Q* : BOOL;
	XV208A_SBRValveR4_CloseCmd AT %Q* : BOOL;
	XV201A_AirBlowerValveR1_CloseCmd AT %Q* : BOOL;
	XV202A_AirBlowerValveR2_CloseCmd AT %Q* : BOOL;
	XV203A_AirBlowerValveR3_CloseCmd AT %Q* : BOOL;
	XV204A_AirBlowerValveR4_CloseCmd AT %Q* : BOOL;
	XV221A_LimeValveR1_CloseCmd AT %Q* : BOOL;
	XV222A_LimeValveR2_CloseCmd AT %Q* : BOOL;
	XV223A_LimeValveR3_CloseCmd AT %Q* : BOOL;
	XV224A_LimeValveR4_CloseCmd AT %Q* : BOOL;
	XV211A_AlumValveR1_CloseCmd AT %Q* : BOOL;
	XV212A_AlumValveR2_CloseCmd AT %Q* : BOOL;
	XV213A_AlumValveR3_CloseCmd AT %Q* : BOOL;
	XV214A_AlumValveR4_CloseCmd AT %Q* : BOOL;
	OPR1AON_ReactorR1_OnlineCmd AT %Q* : BOOL;
	OPR2AON_ReactorR2_OnlineCmd AT %Q* : BOOL;
	OPR3AON_ReactorR3_OnlineCmd AT %Q* : BOOL;
	OPR4AON_ReactorR4_OnlineCmd AT %Q* : BOOL;
	OPR1AOFF_ReactorR1_OfflineCmd AT %Q* : BOOL;
	OPR2AOFF_ReactorR2_OfflineCmd AT %Q* : BOOL;
	OPR3AOFF_ReactorR3_OfflineCmd AT %Q* : BOOL;
	OPR4AOFF_ReactorR4_OfflineCmd AT %Q* : BOOL;
	OPR1ASW_ReactorR1_SwitchCmd AT %Q* : BOOL;
	OPR2ASW_ReactorR2_SwitchCmd AT %Q* : BOOL;
	OPR3ASW_ReactorR3_SwitchCmd AT %Q* : BOOL;
	OPR4ASW_ReactorR4_SwitchCmd AT %Q* : BOOL;
	AUX402_PLCRunStat AT %Q* : BOOL;
	AUX401_CommonAlarm AT %Q* : BOOL;
	LSH201B1_LevelSensorR1 AT %I* : BOOL;
	LSH201B2_LevelSensorR2 AT %I* : BOOL;
	LSH201B3_LevelSensorR3 AT %I* : BOOL;
	LSH201B4_LevelSensorR4 AT %I* : BOOL;
	OPR1B_ReactorStatus AT %I* : BOOL;
	OPR2B_ReactorStatus AT %I* : BOOL;
	OPR3B_ReactorStatus AT %I* : BOOL;
	OPR4B_ReactorStatus AT %I* : BOOL;
	D201B_DoorPanelStatus AT %I* : BOOL;
	F201B_FanStatus AT %I* : BOOL;
	HR201B1_DecantHighLevelR1 AT %I* : BOOL;
	LR201B1_DecantLowLevelR1 AT %I* : BOOL;
	HR201B2_DecantHighLevelR2 AT %I* : BOOL;
	LR201B2_DecantLowLevelR2 AT %I* : BOOL;
	HR201B3_DecantHighLevelR3 AT %I* : BOOL;
	HR201B4_DecantHighLevelR4 AT %I* : BOOL;
	LR201B3_DecantLowLevelR3 AT %I* : BOOL;
	LR201B4_DecantLowLevelR4 AT %I* : BOOL;
	XV205B_SBRValveR1_OpenStat AT %I* : BOOL;
	XV206B_SBRValveR2_OpenStat AT %I* : BOOL;
	XV207B_SBRValveR3_OpenStat AT %I* : BOOL;
	XV208B_SBRValveR4_OpenStat AT %I* : BOOL;
	XV201B_AirBlowerValveR1_OpenStat AT %I* : BOOL;
	XV202B_AirBlowerValveR2_OpenStat AT %I* : BOOL;
	XV203B_AirBlowerValveR3_OpenStat AT %I* : BOOL;
	XV204B_AirBlowerValveR4_OpenStat AT %I* : BOOL;
	XV221B_LimeValveR1_OpenStat AT %I* : BOOL;
	XV222B_LimeValveR2_OpenStat AT %I* : BOOL;
	XV223B_LimeValveR3_OpenStat AT %I* : BOOL;
	XV224B_LimeValveR4_OpenStat AT %I* : BOOL;
	XV211B_AlumValveR1_OpenStat AT %I* : BOOL;
	XV212B_AlumValveR2_OpenStat AT %I* : BOOL;
	XV213B_AlumValveR3_OpenStat AT %I* : BOOL;
	XV214B_AlumValveR4_OpenStat AT %I* : BOOL;
	XV205B_SBRValveR1_CloseStat AT %I* : BOOL;
	XV206B_SBRValveR2_CloseStat AT %I* : BOOL;
	XV207B_SBRValveR3_CloseStat AT %I* : BOOL;
	XV208B_SBRValveR4_CloseStat AT %I* : BOOL;
	XV201B_AirBlowerValveR1_CloseStat AT %I* : BOOL;
	XV202B_AirBlowerValveR2_CloseStat AT %I* : BOOL;
	XV203B_AirBlowerValveR3_CloseStat AT %I* : BOOL;
	XV204B_AirBlowerValveR4_CloseStat AT %I* : BOOL;
	XV221B_LimeValveR1_CloseStat AT %I* : BOOL;
	XV222B_LimeValveR2_CloseStat AT %I* : BOOL;
	XV223B_LimeValveR3_CloseStat AT %I* : BOOL;
	XV224B_LimeValveR4_CloseStat AT %I* : BOOL;
	XV211B_AlumValveR1_CloseStat AT %I* : BOOL;
	XV212B_AlumValveR2_CloseStat AT %I* : BOOL;
	XV213B_AlumValveR3_CloseStat AT %I* : BOOL;
	XV214B_AlumValveR4_CloseStat AT %I* : BOOL;
	XV241B_SludgeValveR1_CloseStat AT %I* : BOOL;
	XV242B_SludgeValveR2_CloseStat AT %I* : BOOL;
	XV243B_SludgeValveR3_CloseStat AT %I* : BOOL;
	XV244B_SludgeValveR4_CloseStat AT %I* : BOOL;
	XV241B_SludgeValveR1_OpenStat AT %I* : BOOL;
	XV242B_SludgeValveR2_OpenStat AT %I* : BOOL;
	XV243B_SludgeValveR3_OpenStat AT %I* : BOOL;
	XV244B_SludgeValveR4_OpenStat AT %I* : BOOL;
	DO201B1_DOProfilesR1: REAL;
	DO201B1_DOProfilesR1_ScaledValue AT%I*:INT;
	DO201B2_DOProfilesR2: REAL;
	DO201B2_DOProfilesR2_ScaledValue AT %I*:INT;
	DO201B3_DOProfilesR3 : REAL;
	DO201B3_DOProfilesR3_ScaledValue AT %I*:INT;
	D0201B4_DOProfilesR4 : REAL;
	D0201B4_DOProfilesR4_ScaledValue AT %I*:INT;
	PHT201B1_pHlevelR1 : REAL;
	PHT201B1_pHlevelR1_ScaledValue AT%I*:INT;
	PHT201B2_pHlevelR2 : REAL;
	PHT201B2_pHlevelR2_ScaledValue AT %I*  :INT;
	PHT201B3_pHlevelR3  : REAL;
	PHT201B3_pHlevelR3_ScaledValue AT %I*:INT;
	PHT201B4_pHlevelR4  : REAL;
	PHT201B4_pHlevelR4_ScaledValue AT %I*:INT;
	XV205B_SBRValveR1_OpenCmd AT %Q* : BOOL;
	XV206B_SBRValveR2_OpenCmd AT %Q* : BOOL;
	XV207B_SBRValveR3_OpenCmd AT %Q* : BOOL;
	XV208B_SBRValveR4_OpenCmd AT %Q* : BOOL;
	XV202B_AirBlowerValveR2_OpenCmd AT %Q* : BOOL;
	XV201B_AirBlowerValveR1_OpenCmd AT %Q* : BOOL;
	XV204B_AirBlowerValveR4_OpenCmd AT %Q* : BOOL;
	XV203B_AirBlowerValveR3_OpenCmd AT %Q* : BOOL;
	XV221B_LimeValveR1_OpenCmd AT %Q* : BOOL;
	XV222B_LimeValveR2_OpenCmd AT %Q* : BOOL;
	XV223B_LimeValveR3_OpenCmd AT %Q* : BOOL;
	XV224B_LimeValveR4_OpenCmd AT %Q* : BOOL;
	XV211B_AlumValveR1_OpenCmd AT %Q* : BOOL;
	XV212B_AlumValveR2_OpenCmd AT %Q* : BOOL;
	XV213B_AlumValveR3_OpenCmd AT %Q* : BOOL;
	XV214B_AlumValveR4_OpenCmd AT %Q* : BOOL;
	XV241B_SludgeValveR1_OpenCmd AT %Q* : BOOL;
	XV242B_SludgeValveR2_OpenCmd AT %Q* : BOOL;
	XV243B_SludgeValveR3_OpenCmd AT %Q* : BOOL;
	XV244B_SludgeValveR4_OpenCmd AT %Q* : BOOL;
	XV241B_SludgeValveR1_CloseCmd AT %Q* : BOOL;
	XV242B_SludgeValveR2_CloseCmd AT %Q* : BOOL;
	XV243B_SludgeValveClosedR3_CloseCmd AT %Q* : BOOL;
	XV244B_SludgeValveR4_CloseCmd AT %Q* : BOOL;
	XV205B_SBRValveR1_CloseCmd AT %Q* : BOOL;
	XV206B_SBRValveR2_CloseCmd AT %Q* : BOOL;
	XV207B_SBRValveR3_CloseCmd AT %Q* : BOOL;
	XV208B_SBRValveR4_CloseCmd AT %Q* : BOOL;
	XV201B_AirBlowerValveR1_CloseCmd AT %Q* : BOOL;
	XV202B_AirBlowerValveR2_CloseCmd AT %Q* : BOOL;
	XV203B_AirBlowerValveR3_CloseCmd AT %Q* : BOOL;
	XV204B_AirBlowerValveR4_CloseCmd AT %Q* : BOOL;
	XV221B_LimeValveR1_CloseCmd AT %Q* : BOOL;
	XV222B_LimeValveR2_CloseCmd AT %Q* : BOOL;
	XV223B_LimeValveR3_CloseCmd AT %Q* : BOOL;
	XV224B_LimeValveR4_CloseCmd AT %Q* : BOOL;
	XV211B_AlumValveR1_CloseCmd AT %Q* : BOOL;
	XV212B_AlumValveR2_CloseCmd AT %Q* : BOOL;
	XV213B_AlumValveR3_CloseCmd AT %Q* : BOOL;
	XV214B_AlumValveR4_CloseCmd AT %Q* : BOOL;
	OPR1BON_ReactorR1_OnlineCmd AT %Q* : BOOL;
	OPR2BON_ReactorR2_OnlineCmd AT %Q* : BOOL;
	OPR3BON_ReactorR3_OnlineCmd AT %Q* : BOOL;
	OPR4BON_ReactorR4_OnlineCmd AT %Q* : BOOL;
	OPR1BOFF_ReactorR1_OfflineCmd AT %Q* : BOOL;
	OPR2BOFF_ReactorR2_OfflineCmd AT %Q* : BOOL;
	OPR3BOFF_ReactorR3_OfflineCmd AT %Q* : BOOL;
	OPR4BOFF_ReactorR4_OfflineCmd AT %Q* : BOOL;
	OPR1BSW_ReactorR1_SwitchCmd AT %Q* : BOOL;
	OPR2BSW_ReactorR2_SwitchCmd AT %Q* : BOOL;
	OPR3BSW_ReactorR3_SwitchCmd AT %Q* : BOOL;
	OPR4BSW_ReactorR4_SwitchCmd AT %Q* : BOOL;
	AUX502_PLCRunStat AT %Q* : BOOL;
	AUX501_CommonAlarm AT %Q* : BOOL;
	LSHH210A_LimeTank1 AT %I* : BOOL;
	LSH210A_LimeTank1 AT %I* : BOOL;
	LSL210A_LimeTank1 AT %I* : BOOL;
	LSD210A_LimeTank1 AT %I* : BOOL;
	LSHH210B_LimeTank2 AT %I* : BOOL;
	LSH210B_LimeTank2 AT %I* : BOOL;
	LSL210B_LimeTank2 AT %I* : BOOL;
	LSD210B_LimeTank2 AT %I* : BOOL;
	LSHH210C_LimeTank3 AT %I* : BOOL;
	LSH210C_LimeTank3 AT %I* : BOOL;
	LSL210C_LimeTank3 AT %I* : BOOL;
	LSD210C_LimeTank3 AT %I* : BOOL;
	LSL351A_AlumTank1 AT %I* : BOOL;
	LSL351B_AlumTank2 AT %I* : BOOL;
	LSL351C_AlumTank3 AT %I* : BOOL;
	LSL351D_AlumTank4 AT %I* : BOOL;
	LSL355A_SodiumHypochloriteTank AT %I* : BOOL;
	LSL355B_SodiumHypochloriteTank AT %I* : BOOL;
	LSL355C_SodiumHypochloriteTank AT %I* : BOOL;
	LSL353A_CausticSodaTank AT %I* : BOOL;
	LSL353B_CausticSodaTank AT %I* : BOOL;
	LSHH301_EffluentSump AT %I* : BOOL;
	LSH301_EffluentSump AT %I* : BOOL;
	LSL301_EffluentSump AT %I* : BOOL;
	LSHH302_CollectionSump AT %I* : BOOL;
	LSH302_CollectionSump AT %I* : BOOL;
	LSL302_CollectionSump AT %I* : BOOL;
	LSH309A_ReUseWaterStorageTank1HIGH AT %I* : BOOL;
	LSH309B_ReUseWaterStorageTank2HIGH AT %I* : BOOL;
	XV251A_LimeSelectorTank_OpenStat AT %I* : BOOL;
	XV251B_LimeSelectorTank_OpenStat AT %I* : BOOL;
	XV251C_LimeSelectorTank_OpenStat AT %I* : BOOL;
	XV251A_LimeSelectorTank_CloseStat AT %I* : BOOL;
	XV251B_LimSelectorTank_CloseStat AT %I* : BOOL;
	XV251C_LimeSelectorTank_CloseStat AT %I* : BOOL;
	OPAlumA_AlumSelectorTank AT %I* : BOOL;
	OPAlumB_AlumSelectorTank AT %I* : BOOL;
	OPAlumC_AlumSelectorTank AT %I* : BOOL;
	OPAlumD_AlumSelectorTank AT %I* : BOOL;
	OPCausticA_CausticSodaSelectorTank1 AT %I* : BOOL;
	OPCausticB_CausticSodaSelectorTank2 AT %I* : BOOL;
	OPSodiumA_SodiumHypochloriteSelectorTank1 AT %I* : BOOL;
	OPSodiumB_SodiumHypochloriteSelectorTank2 AT %I* : BOOL;
	OPSodiumC_SodiumHypochloriteSelectorTank3 AT %I* : BOOL;
	P210A1_LimePumpS1_RunStat AT %I* : BOOL;
	P210A2_LimePumpS1S2_RunStat AT %I* : BOOL;
	P210A3_LimePumpS2_RunStat AT %I* : BOOL;
	P203A_LimeCirculationPump_RunStat AT %I* : BOOL;
	P203B_LimeCirculationPump_RunStat AT %I* : BOOL;
	P211A1_AlumPumpSBRS1_RunStat AT %I* : BOOL;
	P211A2_AlumPumpSBRS1_RunStat AT %I* : BOOL;
	P211B1_AlumPump1SBRS2_RunStat AT %I* : BOOL;
	P211B2_AlumPumpSBRS2_RunStat AT %I* : BOOL;
	P352A_AlumPumpTertiaryDosing_RunStat AT %I* : BOOL;
	P352B_AlumPumpTertiaryDosing_RunStat AT %I* : BOOL;
	XV210A1_LimeValveS1_OpenStat AT %I* : BOOL;
	XV201A2_LimeValveS2_OpenStat AT %I* : BOOL;
	XV210A1_LimeValveS1_CloseStat AT %I* : BOOL;
	XV201A2_LimeValveS2_CloseStat AT %I* : BOOL;
	P354A_CausticSodaPump_RunStat AT %I* : BOOL;
	P354B_CausticSodaPump_RunStat AT %I* : BOOL;
	P356A_SodiumHypochloritePumpChlorinetank_RunStat AT %I* : BOOL;
	P356B_SodiumHypochloritePumpChlorinetank_RunStat AT %I* : BOOL;
	P204A_SodiumHypochloritePumpDisinfectionTank_RunStat AT %I* : BOOL;
	P204B_SodiumHypochloritePumpDisinfectionTank_RunStat AT %I* : BOOL;
	M210A_LimeStirrer_OverloadStat AT %I* : BOOL;
	M210B_LimeStirrer_OverloadStat AT %I* : BOOL;
	M210C_LimeStirrer_OverloadStat AT %I* : BOOL;
	F300_FanStatus AT %I* : BOOL;
	D300_DoorPanelStatus AT %I* : BOOL;
	XV250A_LimeWaterIntakeTank_OpenStat AT %I* : BOOL;
	XV250B_LimeWaterIntakeTank_OpenStat AT %I* : BOOL;
	XV250C_LimeWaterIntakeTank_OpenStat AT %I* : BOOL;
	XV250A_LimeWaterIntakeTank_CloseStat AT %I* : BOOL;
	XV250B_LimeWaterIntakeTank_CloseStat AT %I* : BOOL;
	XV250C_LimeWaterIntakeTank_CloseStat AT %I* : BOOL;
	XV303A_LamellaSludgeDischarge_OpenStat AT %I* : BOOL;
	XV303B_LamellaSludgeDischarge_OpenStat AT %I* : BOOL;
	XV303C_LamellaSludgeDischarge_OpenStat AT %I* : BOOL;
	XV303D_LamellaSludgeDischarge_OpenStat AT %I* : BOOL;
	XV305_TertiaryTreatmentMainValve_OpenStat AT %I* : BOOL;
	XV303A_LamellaSludgeDischarge_CloseStat AT %I* : BOOL;
	XV303B_LamellaSludgeDischarge_CloseStat AT %I* : BOOL;
	XV303C_LamellaSludgeDischarge_CloseStat AT %I* : BOOL;
	XV303D_LamellaSludgeDischarge_CloseStat AT %I* : BOOL;
	XV305_TertiaryTreatmentMainValve_CloseStat AT %I* : BOOL;
	M210A_LimeStirrer_RunStat AT %I* : BOOL;
	M210B_LimeStirrer_RunStat AT %I* : BOOL;
	M210C_LimeStirrer_RunStat AT %I* : BOOL;
	M303A_Floculator_RunStat AT %I* : BOOL;
	M303B_Floculator_RunStat AT %I* : BOOL;
	M303C_Floculator_RunStat AT %I* : BOOL;
	M303D_Floculator_RunStat AT %I* : BOOL;
	P301A_EffluentTransferPump_RunStat AT %I* : BOOL;
	P301B_EffluentTransferPump_RunStat AT %I* : BOOL;
	AUX11_CascadeAerator_OnlineStat:BOOL;
	AUX12_ChlorineAnalyzer_OnlineStat:BOOL;
	P302A_CollectionPump_RunStat AT %I* : BOOL;
	P302B_CollectionPump_RunStat AT %I* : BOOL;
	K301A_AirCompressor_RunStat AT %I* : BOOL;
	K301B_AirCompressor_RunStat AT %I* : BOOL;
	P210A1_LimePumpS1_LocalRemoteStat AT %I* : BOOL;
	P210A2_LimePumpS1_LocalRemoteStat AT %I* : BOOL;
	P210A3_LimePumpS1_LocalRemoteStat AT %I* : BOOL;
	P203A_LimeCirculationPump1_LocalRemoteStat AT %I* : BOOL;
	P203B_LimeCirculationPump2_LocalRemoteStat AT %I* : BOOL;
	P211A1_AlumPumpSBRS1_LocalRemoteStat AT %I* : BOOL;
	P211A2_AlumPumpSBRS1_LocalRemoteStat AT %I* : BOOL;
	P211B1_AlumPumpSBRS2_LocalRemoteStat AT %I* : BOOL;
	P211B2_AlumPump2SBRS2_LocalRemoteStat AT %I* : BOOL;
	P352A_AlumPumpTertiaryDosing_LocalRemoteStat AT %I* : BOOL;
	P352B_AlumPumpTertiaryDosing_LocalRemoteStat AT %I* : BOOL;
	P354A_CausticSodaPump_LocalRemoteStat AT %I* : BOOL;
	P354B_CausticSodaPump_LocalRemoteStat AT %I* : BOOL;
	P356A_SodiumHypochloritePump_LocalRemoteStat AT %I* : BOOL;
	P356B_SodiumHypochloritePump_LocalRemoteStat AT %I* : BOOL;
	P301A_EffluentTransferPump_LocalRemoteStat AT %I* : BOOL;
	P301B_EffluentTransferPump_LocalRemoteStat AT %I* : BOOL;
	P302A_CollectionPump_LocalRemoteStat AT %I* : BOOL;
	P302B_CollectionPump_LocalRemoteStat AT %I* : BOOL;
	K301A_AirCompressor_LocalRemoteStat AT %I* : BOOL;
	K301B_AirCompressor_LocalRemoteStat AT %I* : BOOL;
	M210A_LimeStirrer_LocalRemoteStat AT %I* : BOOL;
	M210B_LimeStirrer_LocalRemoteStat AT %I* : BOOL;
	M210C_LimeStirrer_LocalRemoteStat AT %I* : BOOL;
	P210A1_LimePumpS1_TripStat AT %I* : BOOL;
	P210A2_LimePumpS1_TripStat AT %I* : BOOL;
	P210A3_LimePumpS1_TripStat AT %I* : BOOL;
	P203A_LimeCirculationPump_TripStat AT %I* : BOOL;
	P203B_LimeCirculationPump_TripStat AT %I* : BOOL;
	P211A1_AlumPumpSBRS1_TripStat AT %I* : BOOL;
	P211A2_AlumPumpSBRS1_TripStat AT %I* : BOOL;
	P211B1_AlumPumpSBRS1_TripStat AT %I* : BOOL;
	P211B2_AlumPumpSBRS2_TripStat AT %I* : BOOL;
	P352A_AlumPumpTertiaryDosing_TripStat AT %I* : BOOL;
	P352B_AlumPumpTertiaryDosing_TripStat AT %I* : BOOL;
	P354A_CausticSodaPump_TripStat AT %I* : BOOL;
	P354B_CausticSodaPump_TripStat AT %I* : BOOL;
	P356A_SodiumHypochloritePump_TripStat AT %I* : BOOL;
	P356B_SodiumHypochloritePump_TripStat AT %I* : BOOL;
	P301A_EffluentTransferPump_TripStat AT %I* : BOOL;
	P301B_EffluentTransferPump_TripStat AT %I* : BOOL;
	P302A_CollectionPump_TripStat AT %I* : BOOL;
	P302B_CollectionPump_TripStat AT %I* : BOOL;
	K301A_AirCompressor_TripStat AT %I* : BOOL;
	K301B_AirCompressor_TripStat AT %I* : BOOL;
	M303A_Floculator_TripStat AT %I* : BOOL;
	M303B_Floculator_TripStat AT %I* : BOOL;
	M303C_Floculator_TripStat AT %I* : BOOL;
	M303D_Floculator_TripStat AT %I* : BOOL;
	P210A1_LimePumpS1_EStopStat AT %I* : BOOL;
	P210A2_LimePumpS1_EStopStat AT %I* : BOOL;
	P210A3_LimePumpS1_EStopStat AT %I* : BOOL;
	P203A_LimeCirculationPump_EStopStat AT %I* : BOOL;
	P203B_LimeCirculationPump_EStopStat AT %I* : BOOL;
	P211A1_AlumPumpSBRS1_EStopStat AT %I* : BOOL;
	P211A2_AlumPumpSBRS1_EStopStat AT %I* : BOOL;
	P211B1_AlumPumpSBRS2_EStopStat AT %I* : BOOL;
	P211B2_AlumPumpSBRS2_EStopStat AT %I* : BOOL;
	P352A_AlumPumpTertiaryDosing_EStopStat AT %I* : BOOL;
	P352B_AlumPumpTertiaryDosing_EStopStat AT %I* : BOOL;
	P354A_CausticSodaPump_EStopStat AT %I* : BOOL;
	P354B_CausticSodaPump_EStopStat AT %I* : BOOL;
	P356A_SodiumHypochloritePump_EStopStat AT %I* : BOOL;
	P356B_SodiumHypochloritePump_EStopStat AT %I* : BOOL;
	P301A_EffluentTransferPump_EStopStat AT %I* : BOOL;
	P301B_EffluentTransferPump_EStopStat AT %I* : BOOL;
	P302A_CollectionPump_EStopStat AT %I* : BOOL;
	P302B_CollectionPump_EStopStat AT %I* : BOOL;
	K301A_AirCompressor_EStopStat AT %I* : BOOL;
	K301B_AirCompressor_EStopStat AT %I* : BOOL;
	M210A_LimeStirrer_EStopStat AT %I* : BOOL;
	M210B_LimeStirrer_EStopStat AT %I* : BOOL;
	M210C_LimeStirrer_EStopStat AT %I* : BOOL;
	XV250A_LimeWaterIntakeTank_OpenCmd AT %Q* : BOOL;
	XV250B_LimeWaterIntakeTank_OpenCmd AT %Q* : BOOL;
	XV250C_LimeWaterIntakeTank_OpenCmd AT %Q* : BOOL;
	XV251A_LimeSelectorTank_OpenCmd AT %Q* : BOOL;
	XV251B_LimeSelectorTank_OpenCmd AT %Q* : BOOL;
	XV251C_LimeSelectorTank_OpenCmd AT %Q* : BOOL;
	M210A_LimeStirrer_RunCmd AT %Q* : BOOL;
	M210B_LimeStirrer_RunCmd AT %Q* : BOOL;
	M210C_LimeStirrer_RunCmd AT %Q* : BOOL;
	P210A1_LimePumpS1_RunCmd AT %Q* : BOOL;
	P210A2_LimePumpS1_RunCmd AT %Q* : BOOL;
	P210A3_LimePumpS1_RunCmd AT %Q* : BOOL;
	P210A1_LimeValveS2_OpenCmd AT %Q* : BOOL;
	P210A2_LimeValveS2_OpenCmd AT %Q* : BOOL;
	P354A_CausticSodaPump_RunCmd AT %Q* : BOOL;
	P354B_CausticSodaPump_RunCmd AT %Q* : BOOL;
	P356A_SodiumHypochloritePump_RunCmd AT %Q* : BOOL;
	P356B_SodiumHypochloritePump_RunCmd AT %Q* : BOOL;
	P204A_SodiumHypochloritePump_RunCmd AT %Q* : BOOL;
	P211A1_AlumPumpSBRS1_RunCmd AT %Q* : BOOL;
	P211A2_AlumPumpSBRS1_RunCmd AT %Q* : BOOL;
	P211B1_AlumPumpSBRS2_RunCmd AT %Q* : BOOL;
	P211B2_AlumPumpSBRS2_RunCmd AT %Q* : BOOL;
	P352A_AlumPumpTertiaryDosing_RunCmd AT %Q* : BOOL;
	P352B_AlumPumpTertiaryDosing_RunCmd AT %Q* : BOOL;
	P203A_LimeCirculationPump_RunCmd AT %Q* : BOOL;
	P203B_LimeCirculationPump_RunCmd AT %Q* : BOOL;
	XV303A_LamellaSludgeDischarge_RunCmd AT %Q* : BOOL;
	XV303B_LamellaSludgeDischarge_RunCmd AT %Q* : BOOL;
	XV303C_LamellaSludgeDischarge_RunCmd AT %Q* : BOOL;
	XV303D_LamellaSludgeDischarge_RunCmd AT %Q* : BOOL;
	XV305_TertiaryTreatmentMainValve_OpenCmd AT %Q* : BOOL;
	M303A_Floculator_RunCmd AT %Q* : BOOL;
	M303B_Floculator_RunCmd AT %Q* : BOOL;
	M303C_Floculator_RunCmd AT %Q* : BOOL;
	M303D_Floculator_RunCmd AT %Q* : BOOL;
	P301A_EffluentTransferPump_RunCmd AT %Q* : BOOL;
	P301B_EffluentTransferPump_RunCmd AT %Q* : BOOL;
	P302A_CollectionPump_RunCmd AT %Q* : BOOL;
	P302B_CollectionPump_RunCmd AT %Q* : BOOL;
	K301A_AirCompressor_RunCmd AT %Q* : BOOL;
	K301B_AirCompressor_RunCmd AT %Q* : BOOL;
	AUX1_CirculationOverflow AT %Q* : BOOL;
	AUX2_SystemInletMonitoring AT %Q* : BOOL;
	AUX3_SystemOutletMonitoring AT %Q* : BOOL;
	AUX4_ChlorineHIGH AT %Q* : BOOL;
	AUX5_SBRDosing AT %Q* : BOOL;
	AUX6_ChlorineDosing AT %Q* : BOOL;
	AUX7_DisinfectionDosing AT %Q* : BOOL;
	AUX8_TertiaryDosing AT %Q* : BOOL;
	AUX9_AlumDosing:BOOL;
	AUX10_CausticDosing:BOOL;
	AUX602_PLCRunStat AT %Q* : BOOL;
	AUX601_CommonAlarm AT %Q* : BOOL;
	AUX17_LimeInService AT %Q* : BOOL;
	AUX18_LimeInService AT %Q* : BOOL;
	AUX19_LimeInService AT %Q* : BOOL;
	AUX20_AlumInService AT %Q* : BOOL;
	AUX21_AlumInService AT %Q* : BOOL;
	AUX22_AlumInService AT %Q* : BOOL;
	AUX23_AlumInService AT %Q* : BOOL;
	AUX24_CausticInService AT %Q* : BOOL;
	AUX25_CausticInService AT %Q* : BOOL;
	AUX26_SodiumInService AT %Q* : BOOL;
	AUX27_SodiumInService AT %Q* : BOOL;
	AUX28_SodiumInService AT %Q* : BOOL;
	AUX33_LimeLOW AT %Q* : BOOL;
	AUX34_LimeLOW AT %Q* : BOOL;
	AUX35_LimeLOW AT %Q* : BOOL;
	AUX36_AlumLOW AT %Q* : BOOL;
	AUX37_AlumLOW AT %Q* : BOOL;
	AUX38_AlumLOW AT %Q* : BOOL;
	AUX39_AlumLOW AT %Q* : BOOL;
	AUX40_CausticLOW AT %Q* : BOOL;
	AUX41_CausticLOW AT %Q* : BOOL;
	AUX42_SodiumLOW AT %Q* : BOOL;
	AUX43_SodiumLOW AT %Q* : BOOL;
	AUX44_SodiumLOW AT %Q* : BOOL;
	FT300_EffluentFlowrateEntry: REAL;
	FT300_EffluentFlowrateEntry_ScaledValue AT%I*:INT;
	AT300_EffluentTurbidityEntry : REAL;
	AT300_EffluentTurbidityEntry_ScaledValue AT%I*:INT;
	PHT301_EffluentpHLevelEntry : REAL;
	PHT301_EffluentpHLevelEntry_ScaledValue AT%I*:INT;
	FT301_TreatedEffluentFlowrateDischarge : REAL;
	FT301_TreatedEffluentFlowrateDischarge_ScaledValue AT %I*:INT;
	AT302_TreatedEffluentTurbidityDischarge : REAL;
	AT302_TreatedEffluentTurbidityDischarge_ScaledValue AT %I*:INT;
	PHT303_TreatedEffluentpHLevelDischarge : REAL;
	PHT303_TreatedEffluentpHLevelDischarge_ScaledValue AT%I*:INT;
	CL303_ResidualChlorineAnalyzer : REAL;
	CL303_ResidualChlorineAnalyzer_ScaledValue AT%I*:INT;
	CL304_FinalChlorineAnalyzer : REAL;
	CL304_FinalChlorineAnalyzer_ScaledValue AT%I*:INT;
	ORP_DisinfectionTankAnalyzer : REAL;
	ORP_DisinfectionTankAnalyzer_ScaledValue AT%I*:INT;
	F500_FanStatus AT %I* : BOOL;
	D500_DoorPanelStatus AT %I* : BOOL;
	LSH501A_SludgeStorage AT %I* : BOOL;
	LSHH501A_SludgeStorage AT %I* : BOOL;
	LSL501A_SludgeStorage AT %I* : BOOL;
	LSH501B_SludgeStorage AT %I* : BOOL;
	LSHH501B_SludgeStorage AT %I* : BOOL;
	LSL501B_SludgeStorage AT %I* : BOOL;
	LSH620_FiltrateSumpLevel AT %I* : BOOL;
	LSL620_FiltrateSumpLevel AT %I* : BOOL;
	LSHPU501_PolymerTankLevel AT %I* : BOOL;
	LSLPU501_PolymerTankLevel AT %I* : BOOL;
	PSL505A_PressureSWWaterLine AT %I* : BOOL;
	PSL505B_PressureSWWaterLine2 AT %I* : BOOL;
	P501A_SludgeFeedPump_RunStat AT %I* : BOOL;
	P501B_SludgeFeedPump_RunStat AT %I* : BOOL;
	P501C_SludgeFeedPump_RunStat AT %I* : BOOL;
	B501A_Blower_RunStat AT %I* : BOOL;
	B501B_Blower_RunStat AT %I* : BOOL;
	B501C_Blower_RunStat AT %I* : BOOL;
	M502A_Floculator_RunStat AT %I* : BOOL;
	M502B_Floculator_RunStat AT %I* : BOOL;
	P602A_FiltratePump_RunStat AT %I* : BOOL;
	P602B_FiltratePump_RunStat AT %I* : BOOL;
	XV505A_SolenoidValveLine_OpenStat AT %I* : BOOL;
	XV505B_SolenoidValveLine_OpenStat AT %I* : BOOL;
	XVPU502_DiagpharmAirValve_OpenStat AT %I* : BOOL;
	XV505A_SolenoidValveLine_CloseStat AT %I* : BOOL;
	XV505B_SolenoidValveLine_CloseStat AT %I* : BOOL;
	XVPU502_DiagpharmAirValve_CloseStat AT %I* : BOOL;
	D503A_DrumThickener_RunStat AT %I* : BOOL;
	D503B_DrumThickener_RunStat AT %I* : BOOL;
	P505A_BackwashWaterPump_RunStat AT %I* : BOOL;
	P505B_BackwashWaterPump_RunStat AT %I* : BOOL;
	P505C_BackwashWaterPump_RunStat AT %I* : BOOL;
	XV501A_AirBlowerValve_OpenStat AT %I* : BOOL;
	XV501A_AirBlowerValve_CloseStat AT %I* : BOOL;
	XV501B_AirBlowerValve_OpenStat AT %I* : BOOL;
	XV501B_AirBlowerValve_CloseStat AT %I* : BOOL;
	XVPU501A_PolymerValve_OpenStat AT %I* : BOOL;
	XVPU501A_PolymerValve_CloseStat AT %I* : BOOL;
	XVPU501B_PolymerValve_OpenStat AT %I* : BOOL;
	XVPU501B_PolymerValve_CloseStat AT %I* : BOOL;
	M503_PolymerStirrer_RunStat AT %I* : BOOL;
	XVW501A_WaterValve_OpenStat AT %I* : BOOL;
	XVW501A_WaterValve_CloseStat AT %I* : BOOL;
	B501A_Blower_OverloadStat AT %I* : BOOL;
	B501A_Blower_IncompleteStat AT %I* : BOOL;
	B501B_Blower_OverloadStat AT %I* : BOOL;
	B501B_Blower_IncompleteStat AT %I* : BOOL;
	B501C_Blower_OverloadStat AT %I* : BOOL;
	B501C_Blower_IncompleteStat AT %I* : BOOL;
	P501A_SludgeFeedPump_OverloadStat AT %I* : BOOL;
	P501A_SludgeFeedPump_IncompleteStat AT %I* : BOOL;
	P501B_SludgeFeedPump_OverloadStat AT %I* : BOOL;
	P501B_SludgeFeedPump_IncompleteStat AT %I* : BOOL;
	P501C_SludgeFeedPumpOverloadStat AT %I* : BOOL;
	P501C_SludgeFeedPump_IncompleteStat AT %I* : BOOL;
	P602A_FiltratePump_TripStat AT %I* : BOOL;
	P602B_FiltratePump_TripStat AT %I* : BOOL;
	M502A_Floculator_OverloadStat AT %I* : BOOL;
	M502B_Floculator_OverloadStat AT %I* : BOOL;
	D503A_DrumThickener_OverloadStat AT %I* : BOOL;
	D503B_DrumThickener_OverloadStat AT %I* : BOOL;
	P505A_BackwashWaterPump_OverloadStat AT %I* : BOOL;
	P505B_BackwashWaterPump_OverloadStat AT %I* : BOOL;
	P505C_BackwashWaterPump_OverloadStat AT %I* : BOOL;
	M503_PolymerStirrer_OverloadStat AT %I* : BOOL;
	P501A_SludgeFeedPump_LocalRemoteStat AT %I* : BOOL;
	P501B_SludgeFeedPump_LocalRemoteStat AT %I* : BOOL;
	P501C_SludgeFeedPump_LocalRemoteStat AT %I* : BOOL;
	B501A_Blower_LocalRemoteStat AT %I* : BOOL;
	B501B_Blower_LocalRemoteStat AT %I* : BOOL;
	B501C_Blower_LocalRemoteStat AT %I* : BOOL;
	M502A_Floculator_LocalRemoteStat AT %I* : BOOL;
	M502B_Floculator_LocalRemoteStat AT %I* : BOOL;
	D503A_DrumThickener_LocalRemoteStat AT %I* : BOOL;
	D503B_DrumThickener_LocalRemoteStat AT %I* : BOOL;
	P505A_BackwashWaterPump_LocalRemoteStat AT %I* : BOOL;
	P505B_BackwashWaterPump_LocalRemoteStat AT %I* : BOOL;
	P505C_BackwashWaterPump_LocalRemoteStat AT %I* : BOOL;
	P602A_FiltratePump_LocalRemoteStat AT %I* : BOOL;
	P602B_FiltratePump_LocalRemoteStat AT %I* : BOOL;
	M503_PolymerStirrer_LocalRemoteStat AT %I* : BOOL;
	P501A_SludgeFeedPump_EStopStat AT %I* : BOOL;
	P501B_SludgeFeedPump_EStopStat AT %I* : BOOL;
	P501C_SludgeFeedPump_EStopStat AT %I* : BOOL;
	B501A_Blower_EStopStat AT %I* : BOOL;
	B501B_Blower_EStopStat AT %I* : BOOL;
	B501C_Blower_EStopStat AT %I* : BOOL;
	M502A_Floculator_EStopStat AT %I* : BOOL;
	M502B_Floculator_EStopStat AT %I* : BOOL;
	D503A_DrumThickener_EStopStat AT %I* : BOOL;
	D503B_DrumThickener_EStopStat AT %I* : BOOL;
	P505A_BackwashWaterPump_EStopStat AT %I* : BOOL;
	P505B_BackwashWaterPump_EStopStat AT %I* : BOOL;
	P505C_BackwashWaterPump_EStopStat AT %I* : BOOL;
	P602A_FiltratePump_EStopStat AT %I* : BOOL;
	P602B_FiltratePump_EStopStat AT %I* : BOOL;
	M503_PolymerStirrer_EStopStat AT %I* : BOOL;
	VE801B_SuctionFan_OnOffStat AT %I* : BOOL;
	P802B_CirculationPump_OnOffStat AT %I* : BOOL;
	P803B_CirculationPump_OnOffStat AT %I* : BOOL;
	P804B_CirculationPump_OnOffStat AT %I* : BOOL;
	P805B1_H2S04Pump_OnOffStat AT %I* : BOOL;
	P805B2_H2S04Pump_OnOffStat AT %I* : BOOL;
	P806B1_NAOHPump_OnOffStat AT %I* : BOOL;
	P806B2_NAOHPump_OnOffStat AT %I* : BOOL;
	P807B1_NAOCLPump_OnOffStat AT %I* : BOOL;
	P807B2_NAOCLPump_OnOffStat AT %I* : BOOL;
	VE801B_SuctionFan_OverloadStat AT %I* : BOOL;
	P802B_CirculationPump_OverloadStat AT %I* : BOOL;
	P803B_CirculationPump_OverloadStat AT %I* : BOOL;
	P804B_CirculationPump_OverloadStat AT %I* : BOOL;
	P805B1_H2S04Pump_OverloadStat AT %I* : BOOL;
	P805B2_H2S04Pump_OverloadStat AT %I* : BOOL;
	P806B1_NAOHPump_OverloadStat AT %I* : BOOL;
	P806B2_NAOHPump_OverloadStat AT %I* : BOOL;
	P807B1_NAOCLPump_OverloadStat AT %I* : BOOL;
	P807B2_NAOCLPump_OverloadStat AT %I* : BOOL;
	VE801B_Suction_EStopStat AT %I* : BOOL;
	P802B_CirculationPump_EStopStat AT %I* : BOOL;
	P803B_CirculationPump_EStopStat AT %I* : BOOL;
	P804B_CirculationPump_EStopStat AT %I* : BOOL;
	P805B1_H2S04Pump_EStopStat AT %I* : BOOL;
	P805B2_H2S04Pump_EStopStat AT %I* : BOOL;
	P806B1_NAOHPump_EStopStat AT %I* : BOOL;
	P806B2_NAOHPump_EstopStat AT %I* : BOOL;
	P807B1_NAOCLPump_EStopStat AT %I* : BOOL;
	P807B2_NAOCLPump_EStopStat AT %I* : BOOL;
	LSH600_SludgePitSensor : REAL;
	LSH600_SludgePitSensor_ScaledValue AT%I*:INT;
	XVPU502_DiagpharmAirValve_OpenCmd AT %Q* : BOOL;
	M502A_Floculator_RunCmd AT %Q* : BOOL;
	M502B_Floculator_RunCmd AT %Q* : BOOL;
	D503A_DrumThickener_RunCmd AT %Q* : BOOL;
	D503B_DrumThickener_RunCmd AT %Q* : BOOL;
	P602A_FiltratePump_RunCmd AT %Q* : BOOL;
	P602B_FiltratePump_RunCmd AT %Q* : BOOL;
	XVPU501A_PolymerValve_OpenCloseCmd AT %Q* : BOOL;
	XVPU501B_PolymerValve_OpenCloseCmd AT %Q* : BOOL;
	XV505A_SolenoidValveLine_OpenCmd AT %Q* : BOOL;
	XV505B_SolenoidValveLine_CloseCmd AT %Q* : BOOL;
	XVW501A_WaterValve_OpenCmd AT %Q* : BOOL;
	B501A_Blower_RunCmd AT %Q* : BOOL;
	B501B_Blower_RunCmd AT %Q* : BOOL;
	B501C_Blower_RunCmd AT %Q* : BOOL;
	P501A_SludgeFeedPump_RunCmd AT %Q* : BOOL;
	P501B_SludgeFeedPump_RunCmd AT %Q* : BOOL;
	P501C_SludgeFeedPump_RunCmd AT %Q* : BOOL;
	P505A_BackwashWaterPump_RunCmd AT %Q* : BOOL;
	P505B_BackwashWaterPump_RunCmd AT %Q* : BOOL;
	P505C_BackwashWaterPump_RunCmd AT %Q* : BOOL;
	XV501A_AirBlowerValve_OpenCmd AT %Q* : BOOL;
	XV501B_AirBlowerValve_OpenCmd AT %Q* : BOOL;
	XV501A_AirBlowerValve_CloseCmd AT %Q* : BOOL;
	XV501B_AirBlowerValve_CloseCmd AT %Q* : BOOL;
	M503_PolymerStirrer_FwdCmd AT %Q* : BOOL;
	M503_PolymerStirrer_RvsCmd AT %Q* : BOOL;
	AUX510_SludgeStorageHigh AT %Q* : BOOL;
	AUX511_ReuseWaterStorageLow AT %Q* : BOOL;
	AUX512_FiltrateSumpHigh AT %Q* : BOOL;
	AUX513_SludgePitHigh AT %Q* : BOOL;
	AUX515_SludgePitLow:BOOL;
	AUX514_PolymerLevelLow AT %Q* : BOOL;
	AUX701_CommonAlarm AT %Q* : BOOL;
	AUX702_PLCRunStat AT %Q* : BOOL;
	LSL309A_WaterLevelTank AT %I* : BOOL;
	LSL309B_WaterLevelTank AT %I* : BOOL;
	LSH405_VacuumChestLevel AT %I* : BOOL;
	F400_FanStatus AT %I* : BOOL;
	D400_DoorPanelStatus AT %I* : BOOL;
	FSL101_FreshWaterActivationStatus AT %I* : BOOL;
	PSL412_PressureSwitch AT %I* : BOOL;
	PG413_LowPressureGauge AT %I* : BOOL;
	PG414_HighPressureGauge AT %I* : BOOL;
	XV401_SolenoidValve_OpenStat AT %I* : BOOL;
	XV401_SolenoidValve_CloseStat AT %I* : BOOL;
	P401A_LeadPumpA_OverloadStat AT %I* : BOOL;
	P401A_LeadPumpA_IncompleteStat AT %I* : BOOL;
	P401B_LeadPumpB_OverloadStat AT %I* : BOOL;
	P401B_LeadPumpB_IncompleteStat AT %I* : BOOL;
	P401C_LeadPumpC_OverloadStat AT %I* : BOOL;
	P401C_LeadPumpC_IncompleteStat AT %I* : BOOL;
	P401D_LeadPumpD_OverloadStat AT %I* : BOOL;
	P401D_LeadPumpD_IncompleteStat AT %I* : BOOL;
	P402A_JockeyPumpA_OverloadStat AT %I* : BOOL;
	P402A_JockeyPumpA_IncompleteStat AT %I* : BOOL;
	P402B_JockeyPumpB_OverloadStat AT %I* : BOOL;
	P402B_JockeyPumpB_IncompleteStat AT %I* : BOOL;
	P403A_VacuumPumpA_OverloadStat AT %I* : BOOL;
	P403B_VacuumPumpB_OverloadStat AT %I* : BOOL;
	P401A_LeadPumpA_LocalRemoteStat AT %I* : BOOL;
	P401B_LeadPumpB_LocalRemoteStat AT %I* : BOOL;
	P401C_LeadPumpC_LocalRemoteStat AT %I* : BOOL;
	P401D_LeadPumpD_LocalRemoteStat AT %I* : BOOL;
	P402A_JockeyPumpA_LocalRemoteStat AT %I* : BOOL;
	P402B_JockeyPumpB_LocalRemoteStat AT %I* : BOOL;
	P403A_VacuumPumpA_LocalRemoteStat AT %I* : BOOL;
	P403B_VacuumPumpB_LocalRemoteStat AT %I* : BOOL;
	P401A_LeadPumpA_OnOffStat AT %I* : BOOL;
	P401B_LeadPumpB_OnOffStat AT %I* : BOOL;
	P401C_LeadPumpC_OnOffStat AT %I* : BOOL;
	P401D_LeadPumpD_OnOffStat AT %I* : BOOL;
	P402A_JockeyPumpA_OnOffStat AT %I* : BOOL;
	P402B_JockeyPumpB_OnOffStat AT %I* : BOOL;
	P403A_VacuumPumpA_OnOffStat AT %I* : BOOL;
	P403B_VacuumPumpB_OnOffStat AT %I* : BOOL;
	P401A_LeadPumpA_EStopStat AT %I* : BOOL;
	P401B_LeadPumpB_EStopStat AT %I* : BOOL;
	P401C_LeadPumpC_EStopStat AT %I* : BOOL;
	P401D_LeadPumpD_EStopStat AT %I* : BOOL;
	P402A_JockeyPumpA_EStopStat AT %I* : BOOL;
	P402B_JockeyPumpB_EStopStat AT %I* : BOOL;
	P403A_VacuumPumpA_EStopStat AT %I* : BOOL;
	P403B_VacuumPumpB_EStopStat AT %I* : BOOL;
	XV401_SolenoidValve_OpenCmd AT %Q* : BOOL;
	P401A_LeadPumpA_RunCmd AT %Q* : BOOL;
	P401B_LeadPumpB_RunCmd AT %Q* : BOOL;
	P401C_LeadPumpC_RunCmd AT %Q* : BOOL;
	P401D_LeadPumpD_RunCmd AT %Q* : BOOL;
	P402A_JockeyPumpA_RunCmd AT %Q* : BOOL;
	P402B_JockeyPumpB_RunCmd AT %Q* : BOOL;
	P403A_VacuumPumpA_RunCmd AT %Q* : BOOL;
	P403B_VacuumPumpB_RunCmd AT %Q* : BOOL;
	AUX415_AuxLamp_LowPressure AT %Q* : BOOL;
	AUX416_AuxLamp_TankHighLevel AT %Q* : BOOL;
	AUX417_AuxLamp_SystemPrimed AT %Q* : BOOL;
	AUX801_CommonAlarm AT %Q* : BOOL;
	AUX802_PLCRunStat AT %Q* : BOOL;
	PSL411_PressureTransmitter : REAL;
	PSL411_PressureTransmitter_ScaledValue AT%I*:INT;
	F900_FanStatus AT %I* : BOOL;
	D900_DoorPanelStatus AT %I* : BOOL;
	GENRUN_Generator_RunStat AT %I* : BOOL;
	GENOT_Generator_OverloadStat AT %I* : BOOL;
	GENFAIL_Generator_FailStat AT %I* : BOOL;
	GENESTOP_Generator_EStop_Stat AT %I*:BOOL;
	AUX902_PLCRunStat AT %Q* : BOOL;
	AUX901_CommonAlarm AT %Q* : BOOL;
	AUX903_GeneratorSupplyStat AT %Q* : BOOL;
	AUX904_Stream1_RunStat AT %Q* : BOOL;
	AUX905_Stream2_RunStat AT %Q* : BOOL;
	AUX906_InletWork1_RunStat AT %Q* : BOOL;
	AUX907_BlowerHouse1_RunStat AT %Q* : BOOL;
	AUX908_SBR1_RunStat AT %Q* : BOOL;
	AUX909_InletWork2_RunStat AT %Q* : BOOL;
	AUX910_BlowerHouse2_RunStat AT %Q* : BOOL;
	AUX911_SBR2_RunStat AT %Q* : BOOL;
	AUX912_ChemicalTertiary_RunStat AT %Q* : BOOL;
	AUX913_SludgeThickening_RunStat AT %Q* : BOOL;
	AUX914_FilterPress_RunStat AT %Q* : BOOL;
	AUX915_Reuse_RunStat AT %Q* : BOOL;

(*Koupler Status*)
	ScadaRoom_KouplerUTP_State AT %I*:UINT;
	ScadaRoom_KouplerFiber_State AT %I*:UINT;
	InletWork_1_KouplerFiber_State AT %I*:UINT;
	InletWork_2_KouplerFiber_State AT %I*:UINT;
	BlowerHouse_2_KouplerFiber_State AT %I*:UINT;
	BlowerHouse_1_KouplerFiber_State AT %I*:UINT;
	SBR_1_KouplerFiber_State AT %I*:UINT;
	SBR_2_KouplerFiber_State AT %I*:UINT;
	ChemicalAndTertiary_KouplerFiber_State AT %I*:UINT;
	ChemicalAndTertiary_KouplerUTP_State AT %I*:UINT;
	SludgeThickening_KouplerFiber_State AT %I*:UINT;
	Reused_KouplerFiber_State AT %I*:UINT;
	ScadaRoom_KouplerFiber_Return_State AT %I*:UINT;

	ScadaRoom_KouplerUTP_PortA_StateBool:BOOL;
	ScadaRoom_KouplerFiber_PortA_StateBool:BOOL;
	InletWork_1_KouplerFiber_PortA_StateBool:BOOL;
	InletWork_1_KouplerFiber_PortB_StateBool:BOOL;
	InletWork_2_KouplerUTP_PortA_StateBool:BOOL;
	BlowerHouse_2_KouplerFiber_PortA_StateBool:BOOL;
	BlowerHouse_2_KouplerFiber_PortB_StateBool:BOOL;
	BlowerHouse_1_KouplerUTP_PortA_StateBool:BOOL;
	SBR_1_KouplerFiber_PortA_StateBool:BOOL;
	SBR_1_KouplerFiber_PortB_StateBool:BOOL;
	SBR_2_KouplerFiber_PortA_StateBool:BOOL;
	SBR_2_KouplerFiber_PortB_StateBool:BOOL;
	ChemicalAndTertiary_KouplerFiber_PortA_StateBool:BOOL;
	ChemicalAndTertiary_KouplerFiber_PortB_StateBool:BOOL;
	ChemicalAndTertiary_KouplerUTP_PortA_StateBool:BOOL;
	SludgeThickening_KouplerFiber_PortA_StateBool:BOOL;
	SludgeThickening_KouplerFiber_PortB_StateBool:BOOL;
	Reused_KouplerFiber_PortA_StateBool:BOOL;
	Reused_KouplerFiber_PortB_StateBool:BOOL;
	ScadaRoom_KouplerFiber_PortB_StateBool:BOOL;

(*Reset Button Input*)
(*for machine stall*)
	RST001A_ResetButtonInlet_1 AT %I*:BOOL;
	RST001B_ResetButtonInlet_2 AT %I*:BOOL;
	RST002A_ResetButtonBlowerHouse_1 AT %I*:BOOL;
	RST002B_ResetButtonBlowerHouse_2 AT %I*:BOOL;
	RST003A_ResetButtonSBR_1 AT %I*:BOOL;
	RST003B_ResetButtonSBR_2 AT %I*:BOOL;
	RST004_ResetButtonChemicalTertiary AT %I*:BOOL;
	RST005_ResetButtonSludgeThickening AT %I*:BOOL;
	RST008_ResetButtonReused AT %I*:BOOL;

(*inlet*)
	INLET_A: INLET;
	rA1: BOOL;
	EQUIP_TYPE_1_EQA: EQUIP_TYPE_1;
	r_eqA1: BOOL;
	EQUIP_TYPE_2_MXA: EQUIP_TYPE_2;
	EQUIP_TYPE_3_PSA1: EQUIP_TYPE_3;
	EQUIP_TYPE_3_PSA2: EQUIP_TYPE_3;
	EQUIP_TYPE_4_SCA: EQUIP_TYPE_4;
	EQUIP_TYPE_4_SPA: EQUIP_TYPE_4;
	EQUIP_TYPE_5_CWSA: EQUIP_TYPE_5;
	EQUIP_TYPE_4_FSA1: EQUIP_TYPE_4;
	EQUIP_TYPE_4_FSA2: EQUIP_TYPE_4;
	EQUIP_TYPE_6_WSA1: EQUIP_TYPE_6;
	EQUIP_TYPE_6_WSA2: EQUIP_TYPE_6;
	EQUIP_TYPE_5_GRVA1: EQUIP_TYPE_5;
	EQUIP_TYPE_5_GRVA2: EQUIP_TYPE_5;
	EQUIP_TYPE_4_ClassifierA: EQUIP_TYPE_4;
	EQUP_TYPE_1_STA1: EQUIP_TYPE_1;
	r_STA1: BOOL;


	INLET_B: INLET;
	rB1: BOOL;
	EQUIP_TYPE_1_EQB: EQUIP_TYPE_1;
	r_eqB1: BOOL;
	EQUIP_TYPE_2_MXB: EQUIP_TYPE_2;
	EQUIP_TYPE_3_PSB1: EQUIP_TYPE_3;
	EQUIP_TYPE_3_PSB2: EQUIP_TYPE_3;
	EQUIP_TYPE_4_SCB: EQUIP_TYPE_4;
	EQUIP_TYPE_4_SPB: EQUIP_TYPE_4;
	EQUIP_TYPE_5_CWSB: EQUIP_TYPE_5;
	EQUIP_TYPE_4_FSB1: EQUIP_TYPE_4;
	EQUIP_TYPE_4_FSB2: EQUIP_TYPE_4;
	EQUIP_TYPE_6_WSB1: EQUIP_TYPE_6;
	EQUIP_TYPE_6_WSB2: EQUIP_TYPE_6;
	EQUIP_TYPE_5_GRVB1: EQUIP_TYPE_5;
	EQUIP_TYPE_5_GRVB2: EQUIP_TYPE_5;
	EQUIP_TYPE_4_ClassifierB: EQUIP_TYPE_4;
	EQUP_TYPE_1_STB1: EQUIP_TYPE_1;
	r_STB1: BOOL;

(*inlet blower*)
	EQUP_TYPE_7_Blower: EQUIP_TYPE_7;
	rblower: BOOL;
(*CHEMICAL*)
	CHEMICAL_A: Chemical_new;


	(* UNTUK ADIB LINK*)
	reset_lime_tank_1: BOOL;
	reset_lime_tank_2: BOOL;
	reset_lime_tank_3: BOOL;


	alarm_refillLime_A: BOOL;
	alarm_refillLime_B: BOOL;
	alarm_refillLime_C: BOOL;

	EQUIPMENT_REDUNDANT_AIRBLOWER_P210: EQUIPMENT_REDUNDANT_AIRBLOWER;
	reset_P210: BOOL;

	EQUP_TYPE_1_P211_A: EQUIP_TYPE_1;
	reset_P211_A: BOOL;
	EQUP_TYPE_1_P211_B: EQUIP_TYPE_1;
	reset_P211_B: BOOL;
	EQUP_TYPE_1_P352A: EQUIP_TYPE_1;
	reset_A352: BOOL;
	EQUP_TYPE_1_P354: EQUIP_TYPE_1;
	reset_P354: BOOL;
	EQUP_TYPE_1_P356: EQUIP_TYPE_1;
	reset_P356: BOOL;
	EQUP_TYPE_11_p204: EQUIP_TYPE_11;
	reset_p204: BOOL;

	EQUIP_TYPE_6_XV250A: EQUIP_TYPE_6;
	EQUIP_TYPE_6_XV251A: EQUIP_TYPE_6;
	EQUIP_TYPE_4_M210A: EQUIP_TYPE_4;

	EQUIP_TYPE_6_XV250B: EQUIP_TYPE_6;
	EQUIP_TYPE_6_XV251B: EQUIP_TYPE_6;
	EQUIP_TYPE_4_M210B: EQUIP_TYPE_4;

	EQUIP_TYPE_6_XV250C: EQUIP_TYPE_6;
	EQUIP_TYPE_6_XV251C: EQUIP_TYPE_6;
	EQUIP_TYPE_4_M210C: EQUIP_TYPE_4;


(*SBRA*)
	(*ini adib*)
	alarm_alum_sbr_A1: BOOL;
	alarm_alum_sbr_A2: BOOL;
	alarm_alum_sbr_A3: BOOL;
	alarm_alum_sbr_A4: BOOL;

	resumeAlumA1: BOOL;
	resumealumA2: BOOL;
	resumealumA3: BOOL;
	resumealumA4: BOOL;

	reactorA1: Reactor;
	reactorA2: Reactor;
	reactorA3: Reactor;
	reactorA4: Reactor;

	alum_reactorA1: TIME;
	alum_reactorA2: TIME;
	alum_reactorA3: TIME;
	alum_reactorA4: TIME;

	timeConversion_alumA1 : timeConversion;
	timeConversion_alumA2 : timeConversion;
	timeConversion_alumA3 : timeConversion;
	timeConversion_alumA4 : timeConversion;

	InputTime_alumA1 : WORD;
	InputTime_alumA2 : WORD;
	InputTime_alumA3 : WORD;
	InputTime_alumA4 : WORD;

	OutputTime_alumA1 : WORD;
	OutputTime_alumA2 : WORD;
	OutputTime_alumA3 : WORD;
	OutputTime_alumA4 : WORD;

	fill_selectorA: Fill_selector;
	aerate_selectorA: blower_selector;
	decant_selectorA: Decant_selector;

	EQUIP_TYPE_3_Valva1_RA1: EQUIP_TYPE_9;
	EQUIP_TYPE_8_MIXER_A1: EQUIP_TYPE_8;
	EQUIP_TYPE_3_Valve2_RA1: EQUIP_TYPE_9;
	EQUIP_TYPE_3_Valve3_RA1: EQUIP_TYPE_9;
	EQUIP_TYPE_3_Valve4_RA1: EQUIP_TYPE_9;
	EQUIP_TYPE_9_Valve5_RA1: EQUIP_TYPE_9;
	EQUIP_TYPE_10_Dec_RA1: EQUIP_TYPE_10;
	reset_dec_RA1: BOOL;


	EQUIP_TYPE_3_Valva1_RA2: EQUIP_TYPE_9;
	EQUIP_TYPE_8_MIXER_A2: EQUIP_TYPE_8;
	EQUIP_TYPE_3_Valve2_RA2: EQUIP_TYPE_9;
	EQUIP_TYPE_3_Valve3_RA2: EQUIP_TYPE_9;
	EQUIP_TYPE_3_Valve4_RA2: EQUIP_TYPE_9;
	EQUIP_TYPE_9_Valve5_RA2: EQUIP_TYPE_9;
	EQUIP_TYPE_10_Dec_RA2: EQUIP_TYPE_10;
	reset_dec_RA2: BOOL;


	EQUIP_TYPE_3_Valva1_RA3: EQUIP_TYPE_9;
	EQUIP_TYPE_8_MIXER_A3: EQUIP_TYPE_8;
	EQUIP_TYPE_3_Valve2_RA3: EQUIP_TYPE_9;
	EQUIP_TYPE_3_Valve3_RA3: EQUIP_TYPE_9;
	EQUIP_TYPE_3_Valve4_RA3: EQUIP_TYPE_9;
	EQUIP_TYPE_9_Valve5_RA3: EQUIP_TYPE_9;
	EQUIP_TYPE_10_Dec_RA3: EQUIP_TYPE_10;
	reset_dec_RA3: BOOL;


	EQUIP_TYPE_3_Valva1_RA4: EQUIP_TYPE_9;
	EQUIP_TYPE_8_MIXER_A4: EQUIP_TYPE_8;
	EQUIP_TYPE_3_Valve2_RA4: EQUIP_TYPE_9;
	EQUIP_TYPE_3_Valve3_RA4: EQUIP_TYPE_9;
	EQUIP_TYPE_3_Valve4_RA4: EQUIP_TYPE_9;
	EQUIP_TYPE_9_Valve5_RA4: EQUIP_TYPE_9;
	EQUIP_TYPE_10_Dec_RA4: EQUIP_TYPE_10;
	reset_dec_RA4: BOOL;

	EQUP_TYPE_1_Pump_RA: EQUIP_TYPE_1;
	reset_Pump2_RA: BOOL;

(*SBRB*)


	(*ini adib*)
	alarm_alum_sbr_B1: BOOL;
	alarm_alum_sbr_B2: BOOL;
	alarm_alum_sbr_B3: BOOL;
	alarm_alum_sbr_B4: BOOL;

	reactorB1: Reactor;
	resumeAlumB1: BOOL;

	reactorB2: Reactor;
	resumealumB2: BOOL;


	reactorB3: Reactor;
	resumealumB3: BOOL;


	reactorB4: Reactor;
	resumealumB4: BOOL;


	Alum_reactorB1: TIME;
	alum_reactorB2: TIME;
	alum_reactorB3: TIME;
	alum_reactorB4: TIME;

	timeConversion_alumB1 : timeConversion;
	timeConversion_alumB2 : timeConversion;
	timeConversion_alumB3 : timeConversion;
	timeConversion_alumB4 : timeConversion;

	InputTime_alumB1 : WORD;
	InputTime_alumB2 : WORD;
	InputTime_alumB3 : WORD;
	InputTime_alumB4 : WORD;

	OutputTime_alumB1 : WORD;
	OutputTime_alumB2 : WORD;
	OutputTime_alumB3 : WORD;
	OutputTime_alumB4 : WORD;


	fill_selectorB: Fill_selector;
	aerate_selectorB: blower_selector;
	decant_selectorB: Decant_selector;

	EQUIP_TYPE_3_Valva1_RB1: EQUIP_TYPE_9;
	EQUIP_TYPE_8_MIXER_B1: EQUIP_TYPE_8;
	EQUIP_TYPE_3_Valve2_RB1: EQUIP_TYPE_9;
	EQUIP_TYPE_3_Valve3_RB1: EQUIP_TYPE_9;
	EQUIP_TYPE_3_Valve4_RB1: EQUIP_TYPE_9;
	EQUIP_TYPE_9_Valve5_RB1: EQUIP_TYPE_9;
	EQUIP_TYPE_10_Dec_RB1: EQUIP_TYPE_10;
	reset_dec_RB1: BOOL;


	EQUIP_TYPE_3_Valva1_RB2: EQUIP_TYPE_9;
	EQUIP_TYPE_8_MIXER_B2: EQUIP_TYPE_8;
	EQUIP_TYPE_3_Valve2_RB2: EQUIP_TYPE_9;
	EQUIP_TYPE_3_Valve3_RB2: EQUIP_TYPE_9;
	EQUIP_TYPE_3_Valve4_RB2: EQUIP_TYPE_9;
	EQUIP_TYPE_9_Valve5_RB2: EQUIP_TYPE_9;
	EQUIP_TYPE_10_Dec_RB2: EQUIP_TYPE_10;
	reset_dec_RB2: BOOL;


	EQUIP_TYPE_3_Valva1_RB3: EQUIP_TYPE_9;
	EQUIP_TYPE_8_MIXER_B3: EQUIP_TYPE_8;
	EQUIP_TYPE_3_Valve2_RB3: EQUIP_TYPE_9;
	EQUIP_TYPE_3_Valve3_RB3: EQUIP_TYPE_9;
	EQUIP_TYPE_3_Valve4_RB3: EQUIP_TYPE_9;
	EQUIP_TYPE_9_Valve5_RB3: EQUIP_TYPE_9;
	EQUIP_TYPE_10_Dec_RB3: EQUIP_TYPE_10;
	reset_dec_RB3: BOOL;


	EQUIP_TYPE_3_Valva1_RB4: EQUIP_TYPE_9;
	EQUIP_TYPE_8_MIXER_B4: EQUIP_TYPE_8;
	EQUIP_TYPE_3_Valve2_RB4: EQUIP_TYPE_9;
	EQUIP_TYPE_3_Valve3_RB4: EQUIP_TYPE_9;
	EQUIP_TYPE_3_Valve4_RB4: EQUIP_TYPE_9;
	EQUIP_TYPE_9_Valve5_RB4: EQUIP_TYPE_9;
	EQUIP_TYPE_10_Dec_RB4: EQUIP_TYPE_10;
	reset_dec_RB4: BOOL;

	EQUP_TYPE_1_Pump_RB: EQUIP_TYPE_1;
	reset_Pump2_RB: BOOL;

	sbr_airblower_A: EQUIPMENT_SBR_AIRBLOWER;
	sbr_airblower_B: EQUIPMENT_SBR_AIRBLOWER;

(* sludge holding *)

	sludge_holding_A :sludge_holding;

	EQUIPMENT_REDUNDANT_AIRBLOWER_Sludge1: EQUIPMENT_REDUNDANT_AIRBLOWER;
	EQUIP_TYPE_5_xv501a: EQUIP_TYPE_5;
	EQUIP_TYPE_5_xv501b: EQUIP_TYPE_5;
	EQUIP_TYPE_4_d503: EQUIP_TYPE_4;
	EQUP_TYPE_1_p505: EQUIP_TYPE_1;
	reset_p505: BOOL;
	EQUIP_TYPE_5_xv505A: EQUIP_TYPE_5;
	EQUIP_TYPE_5_xv505B: EQUIP_TYPE_5;
	EQUIP_TYPE_4_M502A: EQUIP_TYPE_4;
	EQUIP_TYPE_4_M502B: EQUIP_TYPE_4;
	EQUIPMENT_REDUNDANT_AIRBLOWER_p501: EQUIPMENT_REDUNDANT_AIRBLOWER;
	EQUIP_TYPE_5_XVPolymerWaterSupply: EQUIP_TYPE_5;
	EQUIP_STIRRER_M503: EQUIP_STIRRER;


	reset_B501: BOOL;
	reset_p501: BOOL;

	alarm_refill_polymer: BOOL;
	reset_polymer: BOOL;


	EQUIP_TYPE_1_P602: EQUIP_TYPE_1;
	reset_P602: BOOL;


	(*tertiary treatment *)
	tertiary_treatment_plant_A: tertiary_treatment_plant;
	reset_tertiary_p301: BOOL;
	reset_tertiary_k301: BOOL;
	reset_tertiary_p302: BOOL;


	EQUP_TYPE_1_P301: EQUIP_TYPE_1;
	EQUIP_TYPE_4_M303A: EQUIP_TYPE_4;
	EQUIP_TYPE_4_M303C: EQUIP_TYPE_4;
	EQUP_TYPE_1_K301: EQUIP_TYPE_1;
	EQUIP_TYPE_5_XV305: EQUIP_TYPE_5;
	EQUP_TYPE_1_p302: EQUIP_TYPE_1;
	EQUIP_TYPE_5_XV303A: EQUIP_TYPE_5;
	EQUIP_TYPE_5_XV303B: EQUIP_TYPE_5;
	EQUIP_TYPE_5_XV303C: EQUIP_TYPE_5;
	EQUIP_TYPE_5_XV303D: EQUIP_TYPE_12;
	EQUIP_TYPE_4_M303B: EQUIP_TYPE_4;


	(*reuse water*)
	REUSE_WATER_A: REUSE_WATER;


	EQUIP_TYPE_2_P402: EQUIP_TYPE_2;
	EQUIP_TYPE_2_P401AB: EQUIP_TYPE_2;
	EQUIP_TYPE_2_P401CD: EQUIP_TYPE_2;
	EQUIP_TYPE_2_P403: EQUIP_TYPE_2;
	EQUIP_TYPE_5_xv401: EQUIP_TYPE_2;


(*
	AlumTime_A1:DWORD;
	AlumTime_A2:DWORD;
	AlumTime_A3:DWORD;
	AlumTime_A4:DWORD;
	AlumTime_B1:DWORD;
	AlumTime_B2:DWORD;
	AlumTime_B3:DWORD;
	AlumTime_B4:DWORD;
*)



	GenActive: BOOL;
	GenFailed: BOOL;

	sbr_reset_A1 AT%I* : BOOL;
	sbr_reset_A2 AT %I*: BOOL;	(*  *)
	sbr_reset_A3 AT %I*: BOOL;	(*  *)
	sbr_reset_A4 AT %I*: BOOL;	(*  *)


	sbr_reset_B1 AT%I* : BOOL;
	sbr_reset_B2 AT %I*: BOOL;	(*  *)
	sbr_reset_B3 AT %I*: BOOL;	(*  *)
	sbr_reset_B4 AT %I*: BOOL;	(*  *)



	Stream_1_2_Inlet_Hold: BOOL;
	hold_desludging_A: BOOL;
	hold_desludging_B: BOOL;
	holdFill_A: BOOL;
	holdFill_B: BOOL;
	hold_tertiary_process: BOOL;
	hold_thickening_process: BOOL;
	hold_inlet_b: BOOL;
	hold_inlet_a: BOOL;
	hold_SBR_A: BOOL;
	hold_SBR_B: BOOL;
	hold_reuse_process: BOOL;
	Reuse_StopAllPump: BOOL;
	Reuse_SystemPrimed: BOOL;
	Reuse_JockeyPump: BOOL;
	Reuse_LeadPumpAB: BOOL;
	Reuse_LeadPumpCD: BOOL;
	Reuse_TON_LineBreak: TON;
	Reuse_CompoundPressureSwitch: BOOL;
	Reuse_VacummPump: BOOL;
END_VAR
reuse_water_ST;
reuse_water_FBD;

(*inlet*)

inlet_mixer;

(*sbr reactor*)
reactorA;
reactorB;


(*CHEMICAL*)
chemical_group;

	
(*sludge holding*)
holding_thickening;

(*tertiary treatment*)
tertiary;

(*reuse water*)
(*reuse_water;*)

(* fallback system*)

GenActive := GENRUN_Generator_RunStat;
GenFailed := GENOT_Generator_OverloadStat OR GENFAIL_Generator_FailStat;

(*Phaselock testing*)
phaselock := TRUE;

hold_desludging_A := hold_desludging_B := (BlowerHouse_2_KouplerFiber_PortA_StateBool AND BlowerHouse_2_KouplerFiber_PortB_StateBool);
hold_tertiary_process := GenFailed OR (ChemicalAndTertiary_KouplerFiber_PortA_StateBool AND ChemicalAndTertiary_KouplerFiber_PortB_StateBool);
hold_thickening_process := GenFailed OR (SludgeThickening_KouplerFiber_PortA_StateBool AND SludgeThickening_KouplerFiber_PortB_StateBool);
hold_inlet_a := (BlowerHouse_2_KouplerFiber_PortA_StateBool AND BlowerHouse_2_KouplerFiber_PortB_StateBool);
hold_inlet_b := GenFailed OR (BlowerHouse_2_KouplerFiber_PortA_StateBool AND BlowerHouse_2_KouplerFiber_PortB_StateBool);
holdFill_A := hold_inlet_a;
holdFill_B := hold_inlet_b;
hold_SBR_A := SBR_1_KouplerFiber_PortA_StateBool AND SBR_1_KouplerFiber_PortB_StateBool;
hold_SBR_B := (SBR_2_KouplerFiber_PortA_StateBool AND SBR_2_KouplerFiber_PortB_StateBool) OR GenActive;
hold_reuse_process := Reused_KouplerFiber_PortA_StateBool AND Reused_KouplerFiber_PortB_StateBool;

(*ANALOG INPUT SCALING VALUE *)
AT300_EffluentTurbidityEntry:=(INT_TO_REAL(AT300_EffluentTurbidityEntry_ScaledValue)/32767.0)*14.0;
AT302_TreatedEffluentTurbidityDischarge:=(INT_TO_REAL(AT302_TreatedEffluentTurbidityDischarge_ScaledValue)/32767.0)*14.0;
CL303_ResidualChlorineAnalyzer:=(INT_TO_REAL(CL303_ResidualChlorineAnalyzer_ScaledValue)/32767.0)*14.0;
CL304_FinalChlorineAnalyzer:=(INT_TO_REAL(CL304_FinalChlorineAnalyzer_ScaledValue)/32767.0)*14.0;
D0201A4_DOProfilesR4:=(INT_TO_REAL(D0201A4_DOProfilesR4_ScaledValue)/32767.0)*14.0;
D0201B4_DOProfilesR4:=(INT_TO_REAL(D0201B4_DOProfilesR4_ScaledValue)/32767.0)*14.0;
DO201A1_DOProfilesR1:=(INT_TO_REAL(DO201A1_DOProfilesR1_ScaledValue)/32767.0)*14.0;
DO201A2_DOProfilesR2:=(INT_TO_REAL(DO201A2_DOProfilesR2_ScaledValue)/32767.0)*14.0;
DO201A3_DOProfilesR3:=(INT_TO_REAL(DO201A3_DOProfilesR3_ScaledValue)/32767.0)*14.0;
DO201B1_DOProfilesR1:=(INT_TO_REAL(DO201B1_DOProfilesR1_ScaledValue)/32767.0)*14.0;
DO201B2_DOProfilesR2:= (INT_TO_REAL(DO201B2_DOProfilesR2_ScaledValue)/32767.0)*14.0;
DO201B3_DOProfilesR3:= (INT_TO_REAL(DO201B3_DOProfilesR3_ScaledValue)/32767.0)*14.0;
FT100A_FlowTotalizerS1:=(INT_TO_REAL(FT100A_FlowTotalizerS1_ScaledValue)/32767.0)*14.0;
FT100B_FlowTotalizerS2:=(INT_TO_REAL(FT100B_FlowTotalizerS2_ScaledValue)/32767.0)*14.0;
FT300_EffluentFlowrateEntry:=(INT_TO_REAL(FT300_EffluentFlowrateEntry_ScaledValue)/32767.0)*14.0;
FT301_TreatedEffluentFlowrateDischarge:=(INT_TO_REAL(FT301_TreatedEffluentFlowrateDischarge_ScaledValue)/32767.0)*14.0;
LSH600_SludgePitSensor:=(INT_TO_REAL(LSH600_SludgePitSensor_ScaledValue)/32767.0)*14.0;
ORP_DisinfectionTankAnalyzer:= (INT_TO_REAL(ORP_DisinfectionTankAnalyzer_ScaledValue)/32767.0)*14.0;
PHT201A1_pHlevelR1:= (INT_TO_REAL(PHT201A1_pHlevelR1_ScaledValue)/32767.0)*14.0;
PHT201A2_pHlevelR2:= (INT_TO_REAL(PHT201A2_pHlevelR2_ScaledValue)/32767.0)*14.0;
PHT201A3_pHlevelR3:=(INT_TO_REAL(PHT201A3_pHlevelR3_ScaledValue)/32767.0)*14.0;
PHT201A4_pHlevelR4:=(INT_TO_REAL(PHT201A4_pHlevelR4_ScaledValue)/32767.0)*14.0;
PHT201B1_pHlevelR1 := (INT_TO_REAL(PHT201B1_pHlevelR1_ScaledValue)/32767.0)*14.0;
PHT201B2_pHlevelR2 := (INT_TO_REAL(PHT201B2_pHlevelR2_ScaledValue)/32767.0)*14.0;
PHT201B3_pHlevelR3 := (INT_TO_REAL(PHT201B3_pHlevelR3_ScaledValue)/32767.0)*14.0;
PHT201B4_pHlevelR4 := (INT_TO_REAL(PHT201B4_pHlevelR4_ScaledValue)/32767.0)*14.0;
PHT301_EffluentpHLevelEntry:=(INT_TO_REAL(PHT301_EffluentpHLevelEntry_ScaledValue)/32767.0)*14.0;
PHT303_TreatedEffluentpHLevelDischarge:=(INT_TO_REAL(PHT303_TreatedEffluentpHLevelDischarge_ScaledValue)/32767.0)*14.0;
PSL411_PressureTransmitter:=(INT_TO_REAL(PSL411_PressureTransmitter_ScaledValue)/32767.0)*16.0;

IF ScadaRoom_KouplerUTP_State=8 THEN
	ScadaRoom_KouplerUTP_PortA_StateBool:=TRUE;
ELSE
	ScadaRoom_KouplerUTP_PortA_StateBool:=FALSE;
END_IF

IF ScadaRoom_KouplerFiber_State=8 THEN
	ScadaRoom_KouplerFiber_PortA_StateBool:=TRUE;
ELSE
	ScadaRoom_KouplerFiber_PortA_StateBool:=FALSE;
END_IF

IF InletWork_1_KouplerFiber_State=5128 THEN(*Port A Failed*)

	InletWork_1_KouplerFiber_PortA_StateBool:=FALSE;
	InletWork_1_KouplerFiber_PortB_StateBool:=TRUE;

ELSIF InletWork_1_KouplerFiber_State=17416 THEN(*Port B Failed*)

	InletWork_1_KouplerFiber_PortA_StateBool:=TRUE;
	InletWork_1_KouplerFiber_PortB_StateBool:=FALSE;

ELSIF InletWork_1_KouplerFiber_State=8 THEN(*Comm OK*)

	InletWork_1_KouplerFiber_PortA_StateBool:=TRUE;
	InletWork_1_KouplerFiber_PortB_StateBool:=TRUE;

ELSE
	InletWork_1_KouplerFiber_PortA_StateBool:=FALSE;
	InletWork_1_KouplerFiber_PortB_StateBool:=FALSE;
END_IF

IF InletWork_2_KouplerFiber_State=8 THEN
	InletWork_2_KouplerUTP_PortA_StateBool:=TRUE;
ELSE
	InletWork_2_KouplerUTP_PortA_StateBool:=FALSE;
END_IF

IF BlowerHouse_2_KouplerFiber_State=5128 THEN(*Port A Failed*)

	BlowerHouse_2_KouplerFiber_PortA_StateBool:=FALSE;
	BlowerHouse_2_KouplerFiber_PortB_StateBool:=TRUE;

ELSIF BlowerHouse_2_KouplerFiber_State=17416 THEN(*Port B Failed*)

	BlowerHouse_2_KouplerFiber_PortA_StateBool:=TRUE;
	BlowerHouse_2_KouplerFiber_PortB_StateBool:=FALSE;

ELSIF BlowerHouse_2_KouplerFiber_State=8 THEN(*Comm OK*)

	BlowerHouse_2_KouplerFiber_PortA_StateBool:=TRUE;
	BlowerHouse_2_KouplerFiber_PortB_StateBool:=TRUE;

ELSE
	BlowerHouse_2_KouplerFiber_PortA_StateBool:=FALSE;
	BlowerHouse_2_KouplerFiber_PortB_StateBool:=FALSE;
END_IF

IF BlowerHouse_1_KouplerFiber_State=8 THEN
	BlowerHouse_1_KouplerUTP_PortA_StateBool:=TRUE;
ELSE
	BlowerHouse_1_KouplerUTP_PortA_StateBool:=FALSE;
END_IF

IF SBR_1_KouplerFiber_State=5128 THEN(*Port A Failed*)

	SBR_1_KouplerFiber_PortA_StateBool:=FALSE;
	SBR_1_KouplerFiber_PortB_StateBool:=TRUE;

ELSIF SBR_1_KouplerFiber_State=17416 THEN(*Port B Failed*)

	SBR_1_KouplerFiber_PortA_StateBool:=TRUE;
	SBR_1_KouplerFiber_PortB_StateBool:=FALSE;

ELSIF SBR_1_KouplerFiber_State=8 THEN(*Comm OK*)

	SBR_1_KouplerFiber_PortA_StateBool:=TRUE;
	SBR_1_KouplerFiber_PortB_StateBool:=TRUE;

ELSE
	SBR_1_KouplerFiber_PortA_StateBool:=FALSE;
	SBR_1_KouplerFiber_PortB_StateBool:=FALSE;
END_IF

IF SBR_2_KouplerFiber_State=5128 THEN(*Port A Failed*)

	SBR_2_KouplerFiber_PortA_StateBool:=FALSE;
	SBR_2_KouplerFiber_PortB_StateBool:=TRUE;

ELSIF SBR_2_KouplerFiber_State=17416 THEN(*Port B Failed*)

	SBR_2_KouplerFiber_PortA_StateBool:=TRUE;
	SBR_2_KouplerFiber_PortB_StateBool:=FALSE;

ELSIF SBR_2_KouplerFiber_State=8 THEN(*Comm OK*)

	SBR_2_KouplerFiber_PortA_StateBool:=TRUE;
	SBR_2_KouplerFiber_PortB_StateBool:=TRUE;

ELSE
	SBR_2_KouplerFiber_PortA_StateBool:=FALSE;
	SBR_2_KouplerFiber_PortB_StateBool:=FALSE;
END_IF

IF ChemicalAndTertiary_KouplerFiber_State=5128 THEN(*Port A Failed*)

	ChemicalAndTertiary_KouplerFiber_PortA_StateBool:=FALSE;
	ChemicalAndTertiary_KouplerFiber_PortB_StateBool:=TRUE;

ELSIF ChemicalAndTertiary_KouplerFiber_State=17416 THEN(*Port B Failed*)

	ChemicalAndTertiary_KouplerFiber_PortA_StateBool:=TRUE;
	ChemicalAndTertiary_KouplerFiber_PortB_StateBool:=FALSE;

ELSIF ChemicalAndTertiary_KouplerFiber_State=8 THEN(*Comm OK*)

	ChemicalAndTertiary_KouplerFiber_PortA_StateBool:=TRUE;
	ChemicalAndTertiary_KouplerFiber_PortB_StateBool:=TRUE;

ELSE
	ChemicalAndTertiary_KouplerFiber_PortA_StateBool:=FALSE;
	ChemicalAndTertiary_KouplerFiber_PortB_StateBool:=FALSE;
END_IF

IF ChemicalAndTertiary_KouplerUTP_State=8 THEN
	ChemicalAndTertiary_KouplerUTP_PortA_StateBool:=TRUE;
ELSE
	ChemicalAndTertiary_KouplerUTP_PortA_StateBool:=FALSE;
END_IF

IF SludgeThickening_KouplerFiber_State=5128 THEN(*Port A Failed*)

	SludgeThickening_KouplerFiber_PortA_StateBool:=FALSE;
	SludgeThickening_KouplerFiber_PortB_StateBool:=TRUE;

ELSIF SludgeThickening_KouplerFiber_State=17416 THEN(*Port B Failed*)

	SludgeThickening_KouplerFiber_PortA_StateBool:=TRUE;
	SludgeThickening_KouplerFiber_PortB_StateBool:=FALSE;

ELSIF SludgeThickening_KouplerFiber_State=8 THEN(*Comm OK*)

	SludgeThickening_KouplerFiber_PortA_StateBool:=TRUE;
	SludgeThickening_KouplerFiber_PortB_StateBool:=TRUE;

ELSE
	SludgeThickening_KouplerFiber_PortA_StateBool:=FALSE;
	SludgeThickening_KouplerFiber_PortB_StateBool:=FALSE;
END_IF

IF Reused_KouplerFiber_State=5128 THEN(*Port A Failed*)

	Reused_KouplerFiber_PortA_StateBool:=FALSE;
	Reused_KouplerFiber_PortB_StateBool:=TRUE;

ELSIF Reused_KouplerFiber_State=17416 THEN(*Port B Failed*)

	Reused_KouplerFiber_PortA_StateBool:=TRUE;
	Reused_KouplerFiber_PortB_StateBool:=FALSE;

ELSIF Reused_KouplerFiber_State=8 THEN(*Comm OK*)

	Reused_KouplerFiber_PortA_StateBool:=TRUE;
	Reused_KouplerFiber_PortB_StateBool:=TRUE;

ELSE
	Reused_KouplerFiber_PortA_StateBool:=FALSE;
	Reused_KouplerFiber_PortB_StateBool:=FALSE;
END_IF

IF ScadaRoom_KouplerFiber_Return_State=8 THEN
	ScadaRoom_KouplerFiber_PortB_StateBool:=TRUE;
ELSE
	ScadaRoom_KouplerFiber_PortB_StateBool:=FALSE;
END_IF

(*INLET STREAM 1 AUXILARY*)
IF LSHH101A_EQFloatSensor THEN
	AUX101A_EQFloatSensor_AlarmS1:=TRUE;
ELSE
	AUX101A_EQFloatSensor_AlarmS1:=FALSE;
END_IF

IF LSHH103A_SBRFloatSensor THEN
	AUX104A_SBRFloatSensor_AlarmS1:=TRUE;
ELSE
	AUX104A_SBRFloatSensor_AlarmS1:=FALSE;
END_IF

IF LSHH105A2_StreamLineOverflow THEN
	AUX105A_StreamSensorOverflow_AlarmS1:=TRUE;
ELSE
	AUX105A_StreamSensorOverflow_AlarmS1:=FALSE;
END_IF

(*INLET STREAM 2 AUXILARY*)
IF LSHH101B_EQFloatSensor THEN
	AUX101B_EQFloatSensor_AlarmS2:=TRUE;
ELSE
	AUX101B_EQFloatSensor_AlarmS2:=FALSE;
END_IF

IF LSHH103B_SBRFloatSensor THEN
	AUX104B_SBRFloatSensor_AlarmS2:=TRUE;
ELSE
	AUX104B_SBRFloatSensor_AlarmS2:=FALSE;
END_IF

IF LSHH105B2_StreamLineOverflow THEN
	AUX105B_StreamSensorOverflow_AlarmS2:=TRUE;
ELSE
	AUX105B_StreamSensorOverflow_AlarmS2:=FALSE;
END_IF

(*BLOWER HOUSE 1 & SBR 1 AUXILARY*)
IF OPR1A_ReactorStatus THEN
	OPR1AON_ReactorR1_OnlineCmd:=TRUE;
	OPR1AOFF_ReactorR1_OfflineCmd:=FALSE;
	AUXA1_ReactorS1R1_OpsStat:=TRUE;
	OPR1ASW_ReactorR1_SwitchCmd:=TRUE;
ELSE
	OPR1AON_ReactorR1_OnlineCmd:=FALSE;
	OPR1AOFF_ReactorR1_OfflineCmd:=TRUE;
	AUXA1_ReactorS1R1_OpsStat:=FALSE;
	OPR1ASW_ReactorR1_SwitchCmd:=FALSE;
END_IF

IF OPR2A_ReactorStatus THEN
	OPR2AON_ReactorR2_OnlineCmd:=TRUE;
	OPR2AOFF_ReactorR2_OfflineCmd:=FALSE;
	AUXA2_ReactorS1R2_OpsStat:=TRUE;
	OPR2ASW_ReactorR2_SwitchCmd:=TRUE;
ELSE
	OPR2AON_ReactorR2_OnlineCmd:=FALSE;
	OPR2AOFF_ReactorR2_OfflineCmd:=TRUE;
	AUXA2_ReactorS1R2_OpsStat:=FALSE;
	OPR2ASW_ReactorR2_SwitchCmd:=FALSE;
END_IF

IF OPR3A_ReactorStatus THEN
	OPR3AON_ReactorR3_OnlineCmd:=TRUE;
	OPR3AOFF_ReactorR3_OfflineCmd:=FALSE;
	AUXA3_ReactorS1R3_OpsStat:=TRUE;
	OPR3ASW_ReactorR3_SwitchCmd:=TRUE;
ELSE
	OPR3AON_ReactorR3_OnlineCmd:=FALSE;
	OPR3AOFF_ReactorR3_OfflineCmd:=TRUE;
	AUXA3_ReactorS1R3_OpsStat:=FALSE;
	OPR3ASW_ReactorR3_SwitchCmd:=FALSE;
END_IF

IF OPR4A_ReactorStatus THEN
	OPR4AON_ReactorR4_OnlineCmd:=TRUE;
	OPR4AOFF_ReactorR4_OfflineCmd:=FALSE;
	AUXA4_ReactorS1R4_OpsStat:=TRUE;
	OPR4ASW_ReactorR4_SwitchCmd:=TRUE;
ELSE
	OPR4AON_ReactorR4_OnlineCmd:=FALSE;
	OPR4AOFF_ReactorR4_OfflineCmd:=TRUE;
	AUXA4_ReactorS1R4_OpsStat:=FALSE;
	OPR4ASW_ReactorR4_SwitchCmd:=FALSE;
END_IF

(*BLOWER HOUSE 2 & SBR 2 AUXILARY*)
IF OPR1B_ReactorStatus THEN
	OPR1BON_ReactorR1_OnlineCmd:=TRUE;
	OPR1BOFF_ReactorR1_OfflineCmd:=FALSE;
	AUXB1_ReactorS2R1_OpsStat:=TRUE;
	OPR1BSW_ReactorR1_SwitchCmd:=TRUE;
ELSE
	OPR1BON_ReactorR1_OnlineCmd:=FALSE;
	OPR1BOFF_ReactorR1_OfflineCmd:=TRUE;
	AUXB1_ReactorS2R1_OpsStat:=FALSE;
	OPR1BSW_ReactorR1_SwitchCmd:=FALSE;
END_IF

IF OPR2B_ReactorStatus THEN
	OPR2BON_ReactorR2_OnlineCmd:=TRUE;
	OPR2BOFF_ReactorR2_OfflineCmd:=FALSE;
	AUXB2_ReactorS2R2_OpsStat:=TRUE;
	OPR2BSW_ReactorR2_SwitchCmd:=TRUE;
ELSE
	OPR2BON_ReactorR2_OnlineCmd:=FALSE;
	OPR2BOFF_ReactorR2_OfflineCmd:=TRUE;
	AUXB2_ReactorS2R2_OpsStat:=FALSE;
	OPR2BSW_ReactorR2_SwitchCmd:=FALSE;
END_IF

IF OPR3B_ReactorStatus THEN
	OPR3BON_ReactorR3_OnlineCmd:=TRUE;
	OPR3BOFF_ReactorR3_OfflineCmd:=FALSE;
	AUXB3_ReactorS2R3_OpsStat:=TRUE;
	OPR3BSW_ReactorR3_SwitchCmd:=TRUE;
ELSE
	OPR3BON_ReactorR3_OnlineCmd:=FALSE;
	OPR3BOFF_ReactorR3_OfflineCmd:=TRUE;
	AUXB3_ReactorS2R3_OpsStat:=FALSE;
	OPR3BSW_ReactorR3_SwitchCmd:=FALSE;
END_IF

IF OPR4B_ReactorStatus THEN
	OPR4BON_ReactorR4_OnlineCmd:=TRUE;
	OPR4BOFF_ReactorR4_OfflineCmd:=FALSE;
	AUXB4_ReactorS2R4_OpsStat:=TRUE;
	OPR4BSW_ReactorR4_SwitchCmd:=TRUE;
ELSE
	OPR4BON_ReactorR4_OnlineCmd:=FALSE;
	OPR4BOFF_ReactorR4_OfflineCmd:=TRUE;
	AUXB4_ReactorS2R4_OpsStat:=FALSE;
	OPR4BSW_ReactorR4_SwitchCmd:=FALSE;
END_IF

IF B201A1_AirBlowerS1_RunStat THEN
	AUXA5_BlowerS1R1:=TRUE;
ELSE
	AUXA5_BlowerS1R1:=FALSE;
END_IF

IF B201A2_AirBlowerS1_RunStat THEN
	AUXA6_BlowerS1R2:=TRUE;
ELSE
	AUXA6_BlowerS1R2:=FALSE;
END_IF

IF B201A3_AirBlowerS1_RunStat THEN
	AUXA7_BlowerS1R3:=TRUE;
ELSE
	AUXA7_BlowerS1R3:=FALSE;
END_IF

IF B201B1_AirBlowerS2_RunStat THEN
	AUXB5_BlowerS2R1:=TRUE;
ELSE
	AUXB5_BlowerS2R1:=FALSE;
END_IF

IF B201B2_AirBlowerS2_RunStat THEN
	AUXB6_BlowerS2R2:=TRUE;
ELSE
	AUXB6_BlowerS2R2:=FALSE;
END_IF

IF B201B2_AirBlowerS2_RunStat THEN
	AUXB7_BlowerS2R3:=TRUE;
ELSE
	AUXB7_BlowerS2R3:=FALSE;
END_IF

(*CHEMICAL AND TERTIARY  AUXILARY*)
IF LSHH302_CollectionSump THEN
	AUX1_CirculationOverflow:=TRUE;
ELSE
	AUX1_CirculationOverflow:=FALSE;
END_IF

IF CL304_FinalChlorineAnalyzer>2.0 THEN(*MORE THAN 2 PPM GIVE ALARM*)
	AUX4_ChlorineHIGH:=TRUE;
ELSE
	AUX4_ChlorineHIGH:=FALSE;
END_IF

IF P211A1_AlumPumpSBRS1_RunStat OR P211A2_AlumPumpSBRS1_RunStat OR P211B1_AlumPump1SBRS2_RunStat OR P211B2_AlumPumpSBRS2_RunStat OR P210A1_LimePumpS1_RunStat OR P210A2_LimePumpS1S2_RunStat OR P210A3_LimePumpS2_RunStat THEN
	AUX5_SBRDosing:=TRUE;
ELSE
	AUX5_SBRDosing:=FALSE;
END_IF

IF P356A_SodiumHypochloritePumpChlorinetank_RunStat OR P356B_SodiumHypochloritePumpChlorinetank_RunStat THEN
	AUX6_ChlorineDosing:=TRUE;
ELSE
	AUX6_ChlorineDosing:=FALSE;
END_IF

IF P204A_SodiumHypochloritePumpDisinfectionTank_RunStat OR P204A_SodiumHypochloritePumpDisinfectionTank_RunStat THEN
	AUX7_DisinfectionDosing:=TRUE;
ELSE
	AUX7_DisinfectionDosing:=FALSE;
END_IF

IF P354A_CausticSodaPump_RunStat OR P354A_CausticSodaPump_RunStat THEN
	AUX8_TertiaryDosing:=TRUE;
	AUX10_CausticDosing:=TRUE;
ELSE
	AUX8_TertiaryDosing:=FALSE;
	AUX10_CausticDosing:=FALSE;
END_IF

IF P352A_AlumPumpTertiaryDosing_RunStat OR P352A_AlumPumpTertiaryDosing_RunStat THEN
	AUX8_TertiaryDosing:=TRUE;
	AUX9_AlumDosing:=TRUE;
ELSE
	AUX8_TertiaryDosing:=FALSE;
	AUX9_AlumDosing:=FALSE;
END_IF

IF XV251A_LimeSelectorTank_OpenStat THEN
	AUX17_LimeInService:=TRUE;
ELSE
	AUX17_LimeInService:=FALSE;
END_IF

IF XV251B_LimeSelectorTank_OpenStat THEN
	AUX18_LimeInService:=TRUE;
ELSE
	AUX18_LimeInService:=FALSE;
END_IF

IF XV251C_LimeSelectorTank_OpenStat THEN
	AUX19_LimeInService:=TRUE;
ELSE
	AUX19_LimeInService:=FALSE;
END_IF

IF OPAlumA_AlumSelectorTank THEN
	AUX20_AlumInService:=TRUE;
ELSE
	AUX20_AlumInService:=FALSE;
END_IF

IF OPAlumB_AlumSelectorTank THEN
	AUX21_AlumInService:=TRUE;
ELSE
	AUX21_AlumInService:=FALSE;
END_IF

IF OPAlumC_AlumSelectorTank THEN
	AUX22_AlumInService:=TRUE;
ELSE
	AUX22_AlumInService:=FALSE;
END_IF

IF OPAlumD_AlumSelectorTank THEN
	AUX23_AlumInService:=TRUE;
ELSE
	AUX23_AlumInService:=FALSE;
END_IF

IF OPCausticA_CausticSodaSelectorTank1 THEN
	AUX24_CausticInService:=TRUE;
ELSE
	AUX24_CausticInService:=FALSE;
END_IF

IF OPCausticB_CausticSodaSelectorTank2 THEN
	AUX25_CausticInService:=TRUE;
ELSE
	AUX25_CausticInService:=FALSE;
END_IF

IF OPSodiumA_SodiumHypochloriteSelectorTank1 THEN
	AUX26_SodiumInService:=TRUE;
ELSE
	AUX26_SodiumInService:=FALSE;
END_IF

IF OPSodiumB_SodiumHypochloriteSelectorTank2 THEN
	AUX27_SodiumInService:=TRUE;
ELSE
	AUX27_SodiumInService:=FALSE;
END_IF

IF OPSodiumC_SodiumHypochloriteSelectorTank3 THEN
	AUX28_SodiumInService:=TRUE;
ELSE
	AUX28_SodiumInService:=FALSE;
END_IF

IF LSL210A_LimeTank1=FALSE THEN
	AUX33_LimeLOW:=TRUE;
ELSE
	AUX33_LimeLOW:=FALSE;
END_IF

IF LSL210B_LimeTank2=FALSE THEN
	AUX34_LimeLOW:=TRUE;
ELSE
	AUX34_LimeLOW:=FALSE;
END_IF

IF LSL210C_LimeTank3=FALSE THEN
	AUX35_LimeLOW:=TRUE;
ELSE
	AUX35_LimeLOW:=FALSE;
END_IF

IF LSL351A_AlumTank1=FALSE THEN
	AUX36_AlumLOW:=TRUE;
ELSE
	AUX36_AlumLOW:=FALSE;
END_IF

IF LSL351B_AlumTank2=FALSE THEN
	AUX37_AlumLOW:=TRUE;
ELSE
	AUX37_AlumLOW:=FALSE;
END_IF

IF LSL351C_AlumTank3=FALSE THEN
	AUX38_AlumLOW:=TRUE;
ELSE
	AUX38_AlumLOW:=FALSE;
END_IF

IF LSL351D_AlumTank4=FALSE THEN
	AUX39_AlumLOW:=TRUE;
ELSE
	AUX39_AlumLOW:=FALSE;
END_IF

IF LSL353A_CausticSodaTank=FALSE THEN
	AUX40_CausticLOW:=TRUE;
ELSE
	AUX40_CausticLOW:=FALSE;
END_IF

IF LSL353B_CausticSodaTank=FALSE THEN
	AUX41_CausticLOW:=TRUE;
ELSE
	AUX41_CausticLOW:=FALSE;
END_IF

IF LSL355A_SodiumHypochloriteTank=FALSE THEN
	AUX42_SodiumLOW:=TRUE;
ELSE
	AUX42_SodiumLOW:=FALSE;
END_IF

IF LSL355B_SodiumHypochloriteTank=FALSE THEN
	AUX43_SodiumLOW:=TRUE;
ELSE
	AUX43_SodiumLOW:=FALSE;
END_IF

IF LSL355C_SodiumHypochloriteTank=FALSE THEN
	AUX44_SodiumLOW:=TRUE;
ELSE
	AUX44_SodiumLOW:=FALSE;
END_IF

(*SLUDGE TCHIKENING AUXILARY*)
IF LSHH501A_SludgeStorage OR LSHH501B_SludgeStorage THEN
	AUX510_SludgeStorageHigh:=TRUE;
ELSE
	AUX510_SludgeStorageHigh:=FALSE;
END_IF

IF LSL309A_WaterLevelTank=FALSE OR LSL309B_WaterLevelTank=FALSE THEN
	AUX511_ReuseWaterStorageLow:=TRUE;
ELSE
	AUX511_ReuseWaterStorageLow:=FALSE;
END_IF

IF LSH620_FiltrateSumpLevel THEN
	AUX512_FiltrateSumpHigh:=TRUE;
ELSE
	AUX512_FiltrateSumpHigh:=FALSE;
END_IF

IF LSH600_SludgePitSensor>1.0 THEN (*MORE THAN 1 METER*)
	AUX513_SludgePitHigh:=TRUE;
ELSE
	AUX513_SludgePitHigh:=FALSE;
END_IF

IF LSH600_SludgePitSensor<=0.0 THEN (*MORE THAN 1 METER*)
	AUX515_SludgePitLow:=TRUE;
ELSE
	AUX515_SludgePitLow:=FALSE;
END_IF

IF LSLPU501_PolymerTankLevel=FALSE THEN
	AUX514_PolymerLevelLow:=TRUE;
ELSE
	AUX514_PolymerLevelLow:=FALSE;
END_IF

(*REUSE SYSTEM AUXILARY*)
IF PSL411_PressureTransmitter<3.5 THEN(*LESS THAN 3.5 BAR*)
	AUX415_AuxLamp_LowPressure:=TRUE;
ELSE
	AUX415_AuxLamp_LowPressure:=FALSE;
END_IF

IF LSH309A_ReUseWaterStorageTank1HIGH OR LSH309B_ReUseWaterStorageTank2HIGH THEN
	AUX416_AuxLamp_TankHighLevel:=TRUE;
ELSE
	AUX416_AuxLamp_TankHighLevel:=FALSE;
END_IF

IF LSH405_VacuumChestLevel THEN
	AUX417_AuxLamp_SystemPrimed:=TRUE;
ELSE
	AUX417_AuxLamp_SystemPrimed:=FALSE;
END_IF

(*SCADA ROOM AUXILARY*)
IF GENRUN_Generator_RunStat=TRUE THEN
	AUX903_GeneratorSupplyStat:=TRUE;
ELSE
	AUX903_GeneratorSupplyStat:=FALSE;
END_IF

IF GENFAIL_Generator_FailStat=TRUE OR GENOT_Generator_OverloadStat=TRUE THEN
	AUX901_CommonAlarm:=TRUE;
END_IF

IF GENFAIL_Generator_FailStat=FALSE AND GENOT_Generator_OverloadStat=FALSE THEN
	AUX901_CommonAlarm:=FALSE;
END_IF

IF LSH105A1_StreamLineFlow OR FT100A_FlowTotalizerS1>1.0 THEN
	AUX904_Stream1_RunStat:=TRUE;
ELSE
	AUX904_Stream1_RunStat:=FALSE;
END_IF

IF LSH105B1_StreamLineFlow OR FT100B_FlowTotalizerS2>1.0 THEN
	AUX905_Stream2_RunStat:=TRUE;
ELSE
	AUX905_Stream2_RunStat:=FALSE;
END_IF

(*PLC RUN STATUS AUXILARY*)
AUX107_PLCRunStat:=TRUE;
AUX202_PLCRunStat:=TRUE;
AUX402_PLCRunStat:=TRUE;
AUX502_PLCRunStat:=TRUE;
AUX602_PLCRunStat:=TRUE;
AUX702_PLCRunStat:=TRUE;
AUX802_PLCRunStat:=TRUE;
AUX902_PLCRunStat:=TRUE;

(*Elcetra Auxilary*)
IF P301A_EffluentTransferPump_RunStat OR P301B_EffluentTransferPump_RunStat THEN
	AUX11_CascadeAerator_OnlineStat:=TRUE;
	AUX12_ChlorineAnalyzer_OnlineStat:=TRUE;
ELSE
	AUX11_CascadeAerator_OnlineStat:=FALSE;
	AUX12_ChlorineAnalyzer_OnlineStat:=FALSE;
END_IF
END_PROGRAM
ACTION chemical_group:
IF NOT hold_tertiary_process THEN
Chemical_A(
	iA1:= LSD210A_LimeTank1,
	iA2:= LSL210A_LimeTank1 ,
	iA3:= LSH210A_LimeTank1,
	iA4:= LSHH210A_LimeTank1,
	rA1:= reset_lime_tank_1,
	iB1:=LSD210B_LimeTank2 ,
	iB2:=LSL210B_LimeTank2 ,
	iB3:=LSH210B_LimeTank2 ,
	iB4:=LSHH210B_LimeTank2 ,
	rB1:=reset_lime_tank_2 ,
	iC1:= LSD210C_LimeTank3,
	iC2:= LSL210C_LimeTank3,
	iC3:= LSH210C_LimeTank3,
	iC4:= LSHH210C_LimeTank3,
	rC1:= reset_lime_tank_3,
	iqA2:= XV251A_LimeSelectorTank_OpenStat,
	iqB2:= XV251B_LimeSelectorTank_OpenStat,
	iqC2:= XV251C_LimeSelectorTank_OpenStat,
	iLRA:=XV221A_LimeValveR1_OpenStat OR XV222A_LimeValveR2_OpenStat OR XV223A_LimeValveR3_OpenStat OR XV224A_LimeValveR4_OpenStat ,
	iLRB:= XV221B_LimeValveR1_OpenStat OR XV222B_LimeValveR2_OpenStat OR XV223B_LimeValveR3_OpenStat OR XV224B_LimeValveR4_OpenStat  ,
	iAop1:= OPAlumA_AlumSelectorTank,
	iAop2:= OPAlumB_AlumSelectorTank,
	iAop3:= OPAlumC_AlumSelectorTank,
	iAop4:= OPAlumD_AlumSelectorTank,
	iAlss1:= LSL351A_AlumTank1,
	iAlss2:= LSL351B_AlumTank2 ,
	iAlss3:=LSL351C_AlumTank3 ,
	iAlss4:=LSL351D_AlumTank4 ,
	iasbrA:=XV211A_AlumValveR1_OpenStat OR XV212A_AlumValveR2_OpenStat OR XV213A_AlumValveR3_OpenStat OR XV214A_AlumValveR4_OpenStat,
	iasbrB:=XV211B_AlumValveR1_OpenStat OR XV212B_AlumValveR2_OpenStat OR XV213B_AlumValveR3_OpenStat OR XV214B_AlumValveR4_OpenStat,
	iCop1:= OPCausticA_CausticSodaSelectorTank1,
	iCop2:= OPCausticB_CausticSodaSelectorTank2,
	ilssC1:= LSL353A_CausticSodaTank,
	ilssC2:= LSL353B_CausticSodaTank,
	itpm:= P301A_EffluentTransferPump_RunStat OR P301B_EffluentTransferPump_RunStat,
	ilssch1:=LSL355A_SodiumHypochloriteTank ,
	ilssch2:=LSL355A_SodiumHypochloriteTank ,
	ilssch3:=LSL355A_SodiumHypochloriteTank ,
	iChop1:= OPSodiumA_SodiumHypochloriteSelectorTank1,
	iChop2:= OPSodiumB_SodiumHypochloriteSelectorTank2,
	iChop3:= OPSodiumC_SodiumHypochloriteSelectorTank3,
	irdAB:= reactorA1.req_decanting OR reactorA2.req_decanting OR reactorA3.req_decanting OR reactorA4.req_decanting OR reactorB1.req_decanting OR reactorB2.req_decanting OR reactorB3.req_decanting OR reactorB4.req_decanting,
	PHT301:=PHT301_EffluentpHLevelEntry,
	CL303:=CL303_ResidualChlorineAnalyzer,
	qA1=> ,
	qA2=> ,
	qA3=> ,
	eA1=> alarm_refillLime_A,
	qB1=> ,
	qB2=> ,
	qB3=> ,
	eB1=>alarm_refillLime_B ,
	qC1=> ,
	qC2=> ,
	qC3=> ,
	eC1=>alarm_refillLime_C ,
	qCir=> ,
	qLA=> , 
	qLB=> ,
	qP1=> ,
	qP2=> ,
	qP3=> ,
	qP4=> ,
	qtA1=> ,
	qtC1=> ,
	qtCH1=> ,
	qdsp=> );
END_IF

EQUIP_TYPE_6_XV250A(
	i1:=NOT Chemical_A.qA1 OR hold_tertiary_process ,
	i2:= Chemical_A.qA2,
	sa1:=XV250A_LimeWaterIntakeTank_CloseStat ,
	sa2:=XV250A_LimeWaterIntakeTank_OpenStat ,
	c1=> ,
	q1=>XV250A_LimeWaterIntakeTank_OpenCmd ,
	e1=> );
EQUIP_TYPE_6_XV251A(
	i1:=NOT Chemical_A.qA2 OR hold_tertiary_process,
	i2:=Chemical_A.qA2 ,
	sa1:= XV251A_LimeSelectorTank_CloseStat,
	sa2:= XV251A_LimeSelectorTank_OpenStat,
	c1=> ,
	q1=>XV251A_LimeSelectorTank_OpenCmd,
	e1=> );
EQUIP_TYPE_4_M210A(
	i1:= NOT Chemical_A.qA3 OR hold_tertiary_process,
	i2:= Chemical_A.qA3 ,
	sa1:=M210A_LimeStirrer_EStopStat ,
	sa2:=M210A_LimeStirrer_LocalRemoteStat,
	sa3:=M210A_LimeStirrer_OverloadStat ,
	sa4:=M210A_LimeStirrer_RunStat ,
	c1=> ,
	q1=> M210A_LimeStirrer_RunCmd ,
	e1=> );

EQUIP_TYPE_6_XV250B(
	i1:=NOT Chemical_A.qB1 OR hold_tertiary_process ,
	i2:= Chemical_A.qB2,
	sa1:=XV250B_LimeWaterIntakeTank_CloseStat ,
	sa2:=XV250B_LimeWaterIntakeTank_OpenStat ,
	c1=> ,
	q1=>XV250B_LimeWaterIntakeTank_OpenCmd ,
	e1=> );
EQUIP_TYPE_6_XV251B(
	i1:=NOT Chemical_A.qB2 OR hold_tertiary_process,
	i2:=Chemical_A.qB2 ,
	sa1:= XV251B_LimSelectorTank_CloseStat,
	sa2:= XV251B_LimeSelectorTank_OpenStat,
	c1=> ,
	q1=>XV251B_LimeSelectorTank_OpenCmd,
	e1=> );
EQUIP_TYPE_4_M210B(
	i1:=NOT Chemical_A.qB3 OR hold_tertiary_process ,
	i2:= Chemical_A.qB3,
	sa1:=M210B_LimeStirrer_EStopStat ,
	sa2:=M210B_LimeStirrer_LocalRemoteStat,
	sa3:=M210B_LimeStirrer_OverloadStat ,
	sa4:=M210B_LimeStirrer_RunStat ,
	c1=> ,
	q1=> M210B_LimeStirrer_RunCmd ,
	e1=> );

EQUIP_TYPE_6_XV250C(
	i1:=NOT Chemical_A.qC1 OR hold_tertiary_process ,
	i2:= Chemical_A.qC2,
	sa1:=XV250C_LimeWaterIntakeTank_CloseStat ,
	sa2:=XV250C_LimeWaterIntakeTank_OpenStat ,
	c1=> ,
	q1=>XV250C_LimeWaterIntakeTank_OpenCmd ,
	e1=> );
EQUIP_TYPE_6_XV251C(
	i1:=NOT Chemical_A.qC2 OR hold_tertiary_process,
	i2:=Chemical_A.qC2 ,
	sa1:= XV251C_LimeSelectorTank_CloseStat,
	sa2:= XV251C_LimeSelectorTank_OpenStat,
	c1=> ,
	q1=>XV251C_LimeSelectorTank_OpenCmd,
	e1=> );
EQUIP_TYPE_4_M210C(
	i1:=NOT Chemical_A.qC3 OR hold_tertiary_process ,
	i2:= Chemical_A.qC3,
	sa1:=M210C_LimeStirrer_EStopStat ,
	sa2:=M210C_LimeStirrer_LocalRemoteStat,
	sa3:=M210C_LimeStirrer_OverloadStat ,
	sa4:=M210C_LimeStirrer_RunStat ,
	c1=> ,
	q1=> M210C_LimeStirrer_RunCmd ,
	e1=> );

EQUIPMENT_REDUNDANT_AIRBLOWER_P210(
	i1 := NOT  Chemical_A.qP1 OR hold_tertiary_process,
	i2 := Chemical_A.qP1,
	i3 := NOT  Chemical_A.qP2 OR hold_tertiary_process,
	i4 := Chemical_A.qP2,
	sa1:=P210A1_LimePumpS1_EStopStat ,
	sa2:= ,
	sa3:=P210A1_LimePumpS1_LocalRemoteStat ,
	sa4:=P210A1_LimePumpS1_TripStat ,
	sa5:=P210A1_LimePumpS1_RunStat,
	sb1:=P210A2_LimePumpS1_EStopStat ,
	sb2:= ,
	sb3:=P210A2_LimePumpS1_LocalRemoteStat ,
	sb4:=P210A2_LimePumpS1_TripStat ,
	sb5:=P210A2_LimePumpS1S2_RunStat ,
	sc1:=P210A3_LimePumpS1_EStopStat ,
	sc2:= ,
	sc3:=P210A3_LimePumpS1_LocalRemoteStat ,
	sc4:=P210A3_LimePumpS1_TripStat ,
	sc5:=P210A3_LimePumpS2_RunStat ,
	q1=>P210A1_LimePumpS1_RunCmd ,
	q2=>P210A2_LimePumpS1_RunCmd ,
	q3=>P210A3_LimePumpS1_RunCmd );


EQUP_TYPE_1_P211_A(
	i1:= NOT Chemical_A.qP3 OR hold_tertiary_process,
	i2:= Chemical_A.qP3,
	r1:=reset_P211_A ,
	sa1:=P211A1_AlumPumpSBRS1_EStopStat ,
	sa2:= ,
	sa3:=P211A1_AlumPumpSBRS1_LocalRemoteStat ,
	sa4:=P211A1_AlumPumpSBRS1_TripStat ,
	sa5:= P211A1_AlumPumpSBRS1_RunStat,
	sb1:= P211A2_AlumPumpSBRS1_EStopStat,
	sb2:= ,
	sb3:=P211A2_AlumPumpSBRS1_LocalRemoteStat ,
	sb4:= P211A2_AlumPumpSBRS1_TripStat,
	sb5:= P211A2_AlumPumpSBRS1_RunStat,
	c1=> ,
	c2=> , 
	q1=>P211A1_AlumPumpSBRS1_RunCmd ,
	q2=>P211A1_AlumPumpSBRS1_RunCmd ,
	e1=> );

EQUP_TYPE_1_P211_B(
	i1:= NOT Chemical_A.qP4 OR hold_tertiary_process,
	i2:= Chemical_A.qP4,
	r1:=reset_P211_B ,
	sa1:=P211B1_AlumPumpSBRS2_EStopStat ,
	sa2:= ,
	sa3:=P211B1_AlumPumpSBRS2_LocalRemoteStat ,
	sa4:=P211B1_AlumPumpSBRS1_TripStat,
	sa5:= P211B1_AlumPump1SBRS2_RunStat,
	sb1:= P211B2_AlumPumpSBRS2_EStopStat,
	sb2:= ,
	sb3:=P211B2_AlumPump2SBRS2_LocalRemoteStat,
	sb4:= P211B2_AlumPumpSBRS2_TripStat,
	sb5:= P211B2_AlumPumpSBRS2_RunStat,
	c1=> ,
	c2=> ,
	q1=>P211B1_AlumPumpSBRS2_RunCmd ,
	q2=>P211B2_AlumPumpSBRS2_RunCmd ,
	e1=> );

EQUP_TYPE_1_P352A(
	i1:=NOT Chemical_A.qtA1 OR hold_tertiary_process ,
	i2:= Chemical_A.qtA1,
	r1:= reset_A352,
	sa1:= P352A_AlumPumpTertiaryDosing_EStopStat,
	sa2:= ,
	sa3:= P352A_AlumPumpTertiaryDosing_LocalRemoteStat,
	sa4:= P352A_AlumPumpTertiaryDosing_TripStat,
	sa5:= P352A_AlumPumpTertiaryDosing_RunStat,
	sb1:= P352B_AlumPumpTertiaryDosing_EStopStat,
	sb2:= ,
	sb3:= P352B_AlumPumpTertiaryDosing_LocalRemoteStat,
	sb4:= P352B_AlumPumpTertiaryDosing_TripStat,
	sb5:= P352B_AlumPumpTertiaryDosing_RunStat,
	c1=> ,
	c2=> , 
	q1=> P352A_AlumPumpTertiaryDosing_RunCmd,
	q2=> P352B_AlumPumpTertiaryDosing_RunCmd,
	e1=> );

EQUP_TYPE_1_P354(
	i1:= NOT Chemical_A.qtC1 OR hold_tertiary_process,
	i2:= Chemical_A.qtC1,
	r1:= reset_P354,
	sa1:=P354A_CausticSodaPump_EStopStat ,
	sa2:= ,
	sa3:=P354A_CausticSodaPump_LocalRemoteStat ,
	sa4:= P354A_CausticSodaPump_TripStat,
	sa5:= P354A_CausticSodaPump_RunStat,
	sb1:= P354B_CausticSodaPump_EStopStat,
	sb2:= ,
	sb3:= P354B_CausticSodaPump_LocalRemoteStat,
	sb4:= P354B_CausticSodaPump_TripStat,
	sb5:= P354B_CausticSodaPump_EStopStat ,
	c1=> ,
	c2=> ,
	q1=> P354A_CausticSodaPump_RunCmd,
	q2=> P354B_CausticSodaPump_RunCmd,
	e1=> );


EQUP_TYPE_1_P356(
	i1:= NOT Chemical_A.qtCH1 OR hold_tertiary_process,
	i2:= Chemical_A.qtCH1,
	r1:= reset_P356,
	sa1:=P356A_SodiumHypochloritePump_EStopStat ,
	sa2:= ,
	sa3:= P356A_SodiumHypochloritePump_LocalRemoteStat,
	sa4:= P356A_SodiumHypochloritePump_TripStat,
	sa5:= P356A_SodiumHypochloritePumpChlorinetank_RunStat,
	sb1:= P356B_SodiumHypochloritePump_EStopStat,
	sb2:= ,
	sb3:=P356B_SodiumHypochloritePump_LocalRemoteStat ,
	sb4:=P356B_SodiumHypochloritePump_TripStat ,
	sb5:= P356B_SodiumHypochloritePumpChlorinetank_RunStat,
	c1=> ,
	c2=> ,
	q1=>P356A_SodiumHypochloritePump_RunCmd ,
	q2=> P356B_SodiumHypochloritePump_RunCmd,
	e1=> );

EQUP_TYPE_11_p204(
	i1:= NOT Chemical_A.qdsp OR hold_tertiary_process,
	i2:= Chemical_A.qdsp,
	sa1:= P204A_SodiumHypochloritePumpDisinfectionTank_RunStat,
	sa2:= P204B_SodiumHypochloritePumpDisinfectionTank_RunStat,
	c1=> ,
	q1=> P204A_SodiumHypochloritePump_RunCmd,
	e1=> );

reset_P211_A := reset_P211_B := reset_A352 := reset_P354 := reset_P356 := RST004_ResetButtonChemicalTertiary;
END_ACTION
ACTION holding_thickening:
IF NOT hold_thickening_process THEN
sludge_holding_A(
	i1A:= LSL501A_SludgeStorage,
	i1B:= LSL501B_SludgeStorage,
	i2A:= LSH501A_SludgeStorage,
	i2B:= LSH501B_SludgeStorage,
	i3A:=LSHH501A_SludgeStorage ,
	i3B:=LSHH501B_SludgeStorage,
	i4:= LSL309A_WaterLevelTank ,
	i5:= LSHPU501_PolymerTankLevel,
	i6:= LSLPU501_PolymerTankLevel,
	i7:= LSH600_SludgePitSensor > 10,
	ic1:=B501A_Blower_RunStat ,
	ic2:= B501C_Blower_RunStat,
	s1:=D503A_DrumThickener_EStopStat OR D503A_DrumThickener_OverloadStat,
	s2:=M503_PolymerStirrer_EStopStat OR M503_PolymerStirrer_OverloadStat ,
	s3:= P505A_BackwashWaterPump_EStopStat OR P505A_BackwashWaterPump_OverloadStat,
	s4:= B501A_Blower_IncompleteStat OR B501A_Blower_OverloadStat OR B501A_Blower_EStopStat,
	s5:= B501B_Blower_IncompleteStat OR B501B_Blower_OverloadStat OR B501B_Blower_EStopStat ,
	if1:=LSL620_FiltrateSumpLevel,
	if2:=LSH620_FiltrateSumpLevel,
	sb1:=LSH103B_SBRFloatSensor,
	sbs1:=P102B1_SBRTransferPump_RunStat OR P102B2_SBRTransferPump_RunStat,
	r1:= reset_polymer,
	q1A=> ,
	q2A=> ,
	q1B=> ,
	q2B=> ,
	q3=> ,
	q4=> ,
	q5=> ,
	q6=> ,
	q7=> ,
	q8=> ,
	q10=> ,
	q11=> ,
	q12=> ,
	q13=> ,
	q14=> ,
	c1=> ,
	e1=>alarm_refill_polymer );
END_IF

EQUIPMENT_REDUNDANT_AIRBLOWER_Sludge1(
	i1:= sludge_holding_A.q1A OR hold_thickening_process,
	i2:= sludge_holding_A.q2A,
	i3:= sludge_holding_A.q1B  OR hold_thickening_process,
	i4:= sludge_holding_A.q2B,
	sa1:=B501A_Blower_EStopStat ,
	sa2:= B501A_Blower_IncompleteStat,
	sa3:= B501A_Blower_LocalRemoteStat,
	sa4:= B501A_Blower_OverloadStat,
	sa5:= B501A_Blower_RunStat,
	sc1:= B501B_Blower_EStopStat,
	sc2:= B501B_Blower_IncompleteStat,
	sc3:= B501B_Blower_LocalRemoteStat,
	sc4:= B501B_Blower_OverloadStat,
	sc5:= B501B_Blower_RunStat,
	sb1:= B501C_Blower_EStopStat,
	sb2:= B501C_Blower_IncompleteStat,
	sb3:= B501C_Blower_LocalRemoteStat,
	sb4:= B501C_Blower_OverloadStat,
	sb5:= B501C_Blower_RunStat,
	r1 := reset_B501,
	q1=> B501A_Blower_RunCmd,
	q2=> B501B_Blower_RunCmd,
	q3=> B501C_Blower_RunCmd,
	e1=>);


